LIN {X 0,Y 315.131,Z 1203.889,A -85,B 0,C 180,E1 20783.16,E2 20783.16} C_VEL
LIN {X 0,Y 315.154,Z 1205.25,A -85,B 0,C 180,E1 20791.453,E2 20791.453} C_VEL
LIN {X 0,Y 316.158,Z 1199.354,A -85,B 0,C 180,E1 20803.96,E2 20803.96} C_VEL
LIN {X 0,Y 324.048,Z 1181.565,A -85,B 0,C 180,E1 20817.292,E2 20817.292} C_VEL
LIN {X 0,Y 343.7,Z 1149.442,A -85,B 0,C 180,E1 20829.889,E2 20829.889} C_VEL
LIN {X 0,Y 371.507,Z 1103.542,A -85,B 0,C 180,E1 20840.099,E2 20840.099} C_VEL
LIN {X 0,Y 400.716,Z 1046.598,A -85,B 0,C 180,E1 20847.513,E2 20847.513} C_VEL
LIN {X 0,Y 425.345,Z 983.768,A -85,B 0,C 180,E1 20852.408,E2 20852.408} C_VEL
LIN {X 0,Y 433.911,Z 955.043,A -85,B 0,C 180,E1 20854.017,E2 20854.017} C_VEL
LIN {X 0,Y 421.498,Z 919.963,A -85,B 0,C 180,E1 20862.12,E2 20862.12} C_VEL
LIN {X 0,Y 420.35,Z 917.292,A -85,B 0,C 180,E1 20862.934,E2 20862.934} C_VEL
LIN {X 0,Y 411.814,Z 911.622,A -85,B 0,C 180,E1 20867.638,E2 20867.638} C_VEL
LIN {X 0,Y 405.611,Z 896.607,A -85,B 0,C 180,E1 20876.721,E2 20876.721} C_VEL
LIN {X 0,Y 405.544,Z 892.791,A -85,B 0,C 180,E1 20883.154,E2 20883.154} C_VEL
LIN {X 0,Y 410.311,Z 905.519,A -85,B 0,C 180,E1 20893.279,E2 20893.279} C_VEL
LIN {X 0,Y 418.579,Z 929.23,A -85,B 0,C 180,E1 20901.755,E2 20901.755} C_VEL
LIN {X 0,Y 422.011,Z 951.384,A -85,B 0,C 180,E1 20906.592,E2 20906.592} C_VEL
LIN {X 0,Y 394.355,Z 1017.185,A -85,B 0,C 180,E1 20911.799,E2 20911.799} C_VEL
LIN {X 0,Y 362.549,Z 1077.585,A -85,B 0,C 180,E1 20919.822,E2 20919.822} C_VEL
LIN {X 0,Y 334.565,Z 1125.328,A -85,B 0,C 180,E1 20930.491,E2 20930.491} C_VEL
LIN {X 0,Y 315.72,Z 1159.766,A -85,B 0,C 180,E1 20943.524,E2 20943.524} C_VEL
LIN {X 0,Y 308.132,Z 1178.996,A -85,B 0,C 180,E1 20957.121,E2 20957.121} C_VEL
LIN {X 0,Y 307.029,Z 1184.767,A -85,B 0,C 180,E1 20968.509,E2 20968.509} C_VEL
LIN {X 0,Y 307.704,Z 1181.392,A -85,B 0,C 180,E1 20979.862,E2 20979.862} C_VEL
LIN {X 0,Y 313.175,Z 1165.32,A -85,B 0,C 180,E1 20993.345,E2 20993.345} C_VEL
LIN {X 0,Y 330.014,Z 1133.188,A -85,B 0,C 180,E1 21006.999,E2 21006.999} C_VEL
LIN {X 0,Y 356.224,Z 1088.459,A -85,B 0,C 180,E1 21018.097,E2 21018.097} C_VEL
LIN {X 0,Y 357.572,Z 1084.641,A -85,B 0,C 180,E1 21018.97,E2 21018.97} C_VEL
LIN {X 0,Y 328.069,Z 1088.331,A -85,B 0,C 180,E1 21024.778,E2 21024.778} C_VEL
LIN {X 0,Y 313.608,Z 1088.004,A -85,B 0,C 180,E1 21030.075,E2 21030.075} C_VEL
LIN {X 0,Y 311.553,Z 1108.151,A -85,B 0,C 180,E1 21037.077,E2 21037.077} C_VEL
LIN {X 0,Y 312.349,Z 1113.298,A -85,B 0,C 180,E1 21044.589,E2 21044.589} C_VEL
LIN {X 0,Y 315.942,Z 1103.128,A -85,B 0,C 180,E1 21051.839,E2 21051.839} C_VEL
LIN {X 0,Y 320.96,Z 1077.982,A -85,B 0,C 180,E1 21058.088,E2 21058.088} C_VEL
LIN {X 0,Y 326.7,Z 1042.871,A -85,B 0,C 180,E1 21062.595,E2 21062.595} C_VEL
LIN {X 0,Y 356.77,Z 1008.219,A -85,B 0,C 180,E1 21067.385,E2 21067.385} C_VEL
LIN {X 0,Y 393.256,Z 951.699,A -85,B 0,C 180,E1 21071.07,E2 21071.07} C_VEL
LIN {X 0,Y 411.965,Z 913.023,A -85,B 0,C 180,E1 21072.823,E2 21072.823} C_VEL
LIN {X 0,Y 423.19,Z 942.489,A -85,B 0,C 180,E1 21081.626,E2 21081.626} C_VEL
LIN {X 0,Y 427.875,Z 961.762,A -85,B 0,C 180,E1 21085.399,E2 21085.399} C_VEL
LIN {X 0,Y 404.101,Z 1028.215,A -85,B 0,C 180,E1 21089.854,E2 21089.854} C_VEL
LIN {X 0,Y 375.524,Z 1086.146,A -85,B 0,C 180,E1 21096.292,E2 21096.292} C_VEL
LIN {X 0,Y 346.004,Z 1135.355,A -85,B 0,C 180,E1 21105.534,E2 21105.534} C_VEL
LIN {X 0,Y 322.579,Z 1171.597,A -85,B 0,C 180,E1 21117.338,E2 21117.338} C_VEL
LIN {X 0,Y 310.478,Z 1193.301,A -85,B 0,C 180,E1 21130.074,E2 21130.074} C_VEL
LIN {X 0,Y 307.152,Z 1203.616,A -85,B 0,C 180,E1 21142.982,E2 21142.982} C_VEL
LIN {X 0,Y 307.154,Z 1204.986,A -85,B 0,C 180,E1 21151.49,E2 21151.49} C_VEL
LIN {X 0,Y 308.235,Z 1199.058,A -85,B 0,C 180,E1 21164.326,E2 21164.326} C_VEL
LIN {X 0,Y 316.646,Z 1181.267,A -85,B 0,C 180,E1 21177.936,E2 21177.936} C_VEL
LIN {X 0,Y 337.284,Z 1148.896,A -85,B 0,C 180,E1 21190.806,E2 21190.806} C_VEL
LIN {X 0,Y 365.305,Z 1104.183,A -85,B 0,C 180,E1 21200.884,E2 21200.884} C_VEL
LIN {X 0,Y 395.451,Z 1047.578,A -85,B 0,C 180,E1 21208.369,E2 21208.369} C_VEL
LIN {X 0,Y 421.317,Z 983.665,A -85,B 0,C 180,E1 21213.363,E2 21213.363} C_VEL
LIN {X 0,Y 428.388,Z 957.756,A -85,B 0,C 180,E1 21215.019,E2 21215.019} C_VEL
LIN {X 0,Y 416.291,Z 922.873,A -85,B 0,C 180,E1 21223.622,E2 21223.622} C_VEL
LIN {X 0,Y 411.814,Z 911.622,A -85,B 0,C 180,E1 21227.638,E2 21227.638} C_VEL
LIN {X 0,Y 405.086,Z 909.3,A -85,B 0,C 180,E1 21232.543,E2 21232.543} C_VEL
LIN {X 0,Y 402.968,Z 900.428,A -85,B 0,C 180,E1 21243.174,E2 21243.174} C_VEL
LIN {X 0,Y 407.499,Z 913.449,A -85,B 0,C 180,E1 21253.392,E2 21253.392} C_VEL
LIN {X 0,Y 414.782,Z 936.697,A -85,B 0,C 180,E1 21261.671,E2 21261.671} C_VEL
LIN {X 0,Y 416.844,Z 956.153,A -85,B 0,C 180,E1 21265.866,E2 21265.866} C_VEL
LIN {X 0,Y 388.043,Z 1021.702,A -85,B 0,C 180,E1 21271.213,E2 21271.213} C_VEL
LIN {X 0,Y 356.34,Z 1079.599,A -85,B 0,C 180,E1 21279.086,E2 21279.086} C_VEL
LIN {X 0,Y 326.739,Z 1127.976,A -85,B 0,C 180,E1 21290.237,E2 21290.237} C_VEL
LIN {X 0,Y 307.623,Z 1161.365,A -85,B 0,C 180,E1 21303.562,E2 21303.562} C_VEL
LIN {X 0,Y 300.218,Z 1179.27,A -85,B 0,C 180,E1 21316.775,E2 21316.775} C_VEL
LIN {X 0,Y 299.031,Z 1185.03,A -85,B 0,C 180,E1 21328.469,E2 21328.469} C_VEL
LIN {X 0,Y 299.733,Z 1181.663,A -85,B 0,C 180,E1 21340.127,E2 21340.127} C_VEL
LIN {X 0,Y 305.639,Z 1165.65,A -85,B 0,C 180,E1 21353.93,E2 21353.93} C_VEL
LIN {X 0,Y 323.692,Z 1133.18,A -85,B 0,C 180,E1 21367.991,E2 21367.991} C_VEL
LIN {X 0,Y 349.387,Z 1090.484,A -85,B 0,C 180,E1 21378.869,E2 21378.869} C_VEL
LIN {X 0,Y 315.361,Z 1093.317,A -85,B 0,C 180,E1 21386.504,E2 21386.504} C_VEL
LIN {X 0,Y 305.321,Z 1093.594,A -85,B 0,C 180,E1 21391.106,E2 21391.106} C_VEL
LIN {X 0,Y 303.549,Z 1110.784,A -85,B 0,C 180,E1 21398.074,E2 21398.074} C_VEL
LIN {X 0,Y 304.837,Z 1114.039,A -85,B 0,C 180,E1 21405.765,E2 21405.765} C_VEL
LIN {X 0,Y 308.957,Z 1102.249,A -85,B 0,C 180,E1 21413.031,E2 21413.031} C_VEL
LIN {X 0,Y 314.302,Z 1075.933,A -85,B 0,C 180,E1 21419.217,E2 21419.217} C_VEL
LIN {X 0,Y 318.593,Z 1052.265,A -85,B 0,C 180,E1 21422.496,E2 21422.496} C_VEL
LIN {X 0,Y 348.177,Z 1021.018,A -85,B 0,C 180,E1 21427.627,E2 21427.627} C_VEL
LIN {X 0,Y 387.366,Z 966.083,A -85,B 0,C 180,E1 21431.617,E2 21431.617} C_VEL
LIN {X 0,Y 410.03,Z 922.736,A -85,B 0,C 180,E1 21433.707,E2 21433.707} C_VEL
LIN {X 0,Y 420.798,Z 954.604,A -85,B 0,C 180,E1 21442.592,E2 21442.592} C_VEL
LIN {X 0,Y 422.833,Z 965.85,A -85,B 0,C 180,E1 21444.637,E2 21444.637} C_VEL
LIN {X 0,Y 397.487,Z 1032.998,A -85,B 0,C 180,E1 21449.295,E2 21449.295} C_VEL
LIN {X 0,Y 367.249,Z 1091.263,A -85,B 0,C 180,E1 21456.091,E2 21456.091} C_VEL
LIN {X 0,Y 336.743,Z 1139.701,A -85,B 0,C 180,E1 21465.796,E2 21465.796} C_VEL
LIN {X 0,Y 313.19,Z 1174.637,A -85,B 0,C 180,E1 21478.126,E2 21478.126} C_VEL
LIN {X 0,Y 301.461,Z 1195.76,A -85,B 0,C 180,E1 21492.07,E2 21492.07} C_VEL
LIN {X 0,Y 299.108,Z 1204.275,A -85,B 0,C 180,E1 21505.713,E2 21505.713} C_VEL
LIN {X 0,Y 299.153,Z 1203.069,A -85,B 0,C 180,E1 21517.906,E2 21517.906} C_VEL
LIN {X 0,Y 303.852,Z 1190.722,A -85,B 0,C 180,E1 21532.295,E2 21532.295} C_VEL
LIN {X 0,Y 320.169,Z 1164.103,A -85,B 0,C 180,E1 21546.417,E2 21546.417} C_VEL
LIN {X 0,Y 346.421,Z 1124.982,A -85,B 0,C 180,E1 21557.756,E2 21557.756} C_VEL
LIN {X 0,Y 376.502,Z 1074.926,A -85,B 0,C 180,E1 21566.192,E2 21566.192} C_VEL
LIN {X 0,Y 405.351,Z 1014.417,A -85,B 0,C 180,E1 21572.292,E2 21572.292} C_VEL
LIN {X 0,Y 423.592,Z 962.674,A -85,B 0,C 180,E1 21575.609,E2 21575.609} C_VEL
LIN {X 0,Y 412.761,Z 929.669,A -85,B 0,C 180,E1 21583.933,E2 21583.933} C_VEL
LIN {X 0,Y 405.086,Z 909.3,A -85,B 0,C 180,E1 21592.543,E2 21592.543} C_VEL
LIN {X 0,Y 400.156,Z 911.018,A -85,B 0,C 180,E1 21597.565,E2 21597.565} C_VEL
LIN {X 0,Y 400.518,Z 908.117,A -85,B 0,C 180,E1 21603.194,E2 21603.194} C_VEL
LIN {X 0,Y 404.248,Z 920.191,A -85,B 0,C 180,E1 21612.95,E2 21612.95} C_VEL
LIN {X 0,Y 410.57,Z 942.627,A -85,B 0,C 180,E1 21621.209,E2 21621.209} C_VEL
LIN {X 0,Y 412.177,Z 959.739,A -85,B 0,C 180,E1 21625.055,E2 21625.055} C_VEL
LIN {X 0,Y 382.094,Z 1025.525,A -85,B 0,C 180,E1 21630.529,E2 21630.529} C_VEL
LIN {X 0,Y 348.928,Z 1083.517,A -85,B 0,C 180,E1 21638.686,E2 21638.686} C_VEL
LIN {X 0,Y 318.994,Z 1130.538,A -85,B 0,C 180,E1 21649.954,E2 21649.954} C_VEL
LIN {X 0,Y 299.513,Z 1162.965,A -85,B 0,C 180,E1 21663.601,E2 21663.601} C_VEL
LIN {X 0,Y 292.316,Z 1179.544,A -85,B 0,C 180,E1 21676.411,E2 21676.411} C_VEL
LIN {X 0,Y 291.041,Z 1185.293,A -85,B 0,C 180,E1 21688.427,E2 21688.427} C_VEL
LIN {X 0,Y 291.769,Z 1181.936,A -85,B 0,C 180,E1 21700.407,E2 21700.407} C_VEL
LIN {X 0,Y 297.561,Z 1166.965,A -85,B 0,C 180,E1 21713.902,E2 21713.902} C_VEL
LIN {X 0,Y 315.642,Z 1135.83,A -85,B 0,C 180,E1 21728.142,E2 21728.142} C_VEL
LIN {X 0,Y 339.978,Z 1096.243,A -85,B 0,C 180,E1 21738.919,E2 21738.919} C_VEL
LIN {X 0,Y 310.182,Z 1098.354,A -85,B 0,C 180,E1 21745.869,E2 21745.869} C_VEL
LIN {X 0,Y 296.873,Z 1098.049,A -85,B 0,C 180,E1 21752.042,E2 21752.042} C_VEL
LIN {X 0,Y 295.59,Z 1112.991,A -85,B 0,C 180,E1 21759.035,E2 21759.035} C_VEL
LIN {X 0,Y 297.337,Z 1114.841,A -85,B 0,C 180,E1 21766.813,E2 21766.813} C_VEL
LIN {X 0,Y 302.125,Z 1101.315,A -85,B 0,C 180,E1 21774.32,E2 21774.32} C_VEL
LIN {X 0,Y 307.885,Z 1073.731,A -85,B 0,C 180,E1 21780.436,E2 21780.436} C_VEL
LIN {X 0,Y 311.61,Z 1060.112,A -85,B 0,C 180,E1 21782.66,E2 21782.66} C_VEL
LIN {X 0,Y 343.879,Z 1028.138,A -85,B 0,C 180,E1 21788.412,E2 21788.412} C_VEL
LIN {X 0,Y 384.153,Z 974.953,A -85,B 0,C 180,E1 21792.405,E2 21792.405} C_VEL
LIN {X 0,Y 407.556,Z 932.261,A -85,B 0,C 180,E1 21794.343,E2 21794.343} C_VEL
LIN {X 0,Y 417.432,Z 963.741,A -85,B 0,C 180,E1 21802.883,E2 21802.883} C_VEL
LIN {X 0,Y 417.409,Z 971.066,A -85,B 0,C 180,E1 21803.924,E2 21803.924} C_VEL
LIN {X 0,Y 390.801,Z 1037.652,A -85,B 0,C 180,E1 21808.729,E2 21808.729} C_VEL
LIN {X 0,Y 359.742,Z 1094.763,A -85,B 0,C 180,E1 21815.667,E2 21815.667} C_VEL
LIN {X 0,Y 328.906,Z 1141.72,A -85,B 0,C 180,E1 21825.471,E2 21825.471} C_VEL
LIN {X 0,Y 304.384,Z 1176.732,A -85,B 0,C 180,E1 21838.527,E2 21838.527} C_VEL
LIN {X 0,Y 293.483,Z 1195.888,A -85,B 0,C 180,E1 21852.011,E2 21852.011} C_VEL
LIN {X 0,Y 291.097,Z 1204.007,A -85,B 0,C 180,E1 21865.595,E2 21865.595} C_VEL
LIN {X 0,Y 291.163,Z 1203.01,A -85,B 0,C 180,E1 21877.566,E2 21877.566} C_VEL
LIN {X 0,Y 295.159,Z 1192.452,A -85,B 0,C 180,E1 21891.175,E2 21891.175} C_VEL
LIN {X 0,Y 310.316,Z 1168.09,A -85,B 0,C 180,E1 21905.499,E2 21905.499} C_VEL
LIN {X 0,Y 337.055,Z 1129.942,A -85,B 0,C 180,E1 21917.545,E2 21917.545} C_VEL
LIN {X 0,Y 368.849,Z 1079.537,A -85,B 0,C 180,E1 21926.579,E2 21926.579} C_VEL
LIN {X 0,Y 399.806,Z 1017.759,A -85,B 0,C 180,E1 21933.031,E2 21933.031} C_VEL
LIN {X 0,Y 418.696,Z 967.227,A -85,B 0,C 180,E1 21936.303,E2 21936.303} C_VEL
LIN {X 0,Y 408.498,Z 934.625,A -85,B 0,C 180,E1 21944.866,E2 21944.866} C_VEL
LIN {X 0,Y 401.343,Z 913.898,A -85,B 0,C 180,E1 21954.513,E2 21954.513} C_VEL
LIN {X 0,Y 400.156,Z 911.018,A -85,B 0,C 180,E1 21957.565,E2 21957.565} C_VEL
LIN {X 0,Y 397.67,Z 915.644,A -85,B 0,C 180,E1 21962.65,E2 21962.65} C_VEL
LIN {X 0,Y 400.781,Z 926.844,A -85,B 0,C 180,E1 21972.508,E2 21972.508} C_VEL
LIN {X 0,Y 406.304,Z 948.436,A -85,B 0,C 180,E1 21980.711,E2 21980.711} C_VEL
LIN {X 0,Y 407.109,Z 964.414,A -85,B 0,C 180,E1 21984.297,E2 21984.297} C_VEL
LIN {X 0,Y 375.809,Z 1030.127,A -85,B 0,C 180,E1 21989.909,E2 21989.909} C_VEL
LIN {X 0,Y 341.819,Z 1086.973,A -85,B 0,C 180,E1 21998.178,E2 21998.178} C_VEL
LIN {X 0,Y 311.225,Z 1132.932,A -85,B 0,C 180,E1 22009.663,E2 22009.663} C_VEL
LIN {X 0,Y 291.412,Z 1164.556,A -85,B 0,C 180,E1 22023.643,E2 22023.643} C_VEL
LIN {X 0,Y 284.061,Z 1181.005,A -85,B 0,C 180,E1 22037.58,E2 22037.58} C_VEL
LIN {X 0,Y 283.042,Z 1185.556,A -85,B 0,C 180,E1 22048.383,E2 22048.383} C_VEL
LIN {X 0,Y 283.837,Z 1182.208,A -85,B 0,C 180,E1 22060.701,E2 22060.701} C_VEL
LIN {X 0,Y 290.254,Z 1166.966,A -85,B 0,C 180,E1 22074.758,E2 22074.758} C_VEL
LIN {X 0,Y 309.907,Z 1135.149,A -85,B 0,C 180,E1 22089.434,E2 22089.434} C_VEL
LIN {X 0,Y 331.577,Z 1102.546,A -85,B 0,C 180,E1 22098.535,E2 22098.535} C_VEL
LIN {X 0,Y 292.123,Z 1101.841,A -85,B 0,C 180,E1 22110.535,E2 22110.535} C_VEL
LIN {X 0,Y 288.505,Z 1102.454,A -85,B 0,C 180,E1 22113.114,E2 22113.114} C_VEL
LIN {X 0,Y 287.724,Z 1115.062,A -85,B 0,C 180,E1 22120.049,E2 22120.049} C_VEL
LIN {X 0,Y 289.979,Z 1115.281,A -85,B 0,C 180,E1 22128.009,E2 22128.009} C_VEL
LIN {X 0,Y 295.095,Z 1101.275,A -85,B 0,C 180,E1 22135.294,E2 22135.294} C_VEL
LIN {X 0,Y 301.281,Z 1073.043,A -85,B 0,C 180,E1 22141.443,E2 22141.443} C_VEL
LIN {X 0,Y 332.801,Z 1041.917,A -85,B 0,C 180,E1 22148.307,E2 22148.307} C_VEL
LIN {X 0,Y 370.527,Z 998.297,A -85,B 0,C 180,E1 22152.317,E2 22152.317} C_VEL
LIN {X 0,Y 405.129,Z 942.403,A -85,B 0,C 180,E1 22155.152,E2 22155.152} C_VEL
LIN {X 0,Y 413.383,Z 971.51,A -85,B 0,C 180,E1 22162.877,E2 22162.877} C_VEL
LIN {X 0,Y 385.674,Z 1039.157,A -85,B 0,C 180,E1 22167.852,E2 22167.852} C_VEL
LIN {X 0,Y 353.683,Z 1095.936,A -85,B 0,C 180,E1 22174.854,E2 22174.854} C_VEL
LIN {X 0,Y 321.493,Z 1143.165,A -85,B 0,C 180,E1 22184.97,E2 22184.97} C_VEL
LIN {X 0,Y 297.302,Z 1176.315,A -85,B 0,C 180,E1 22197.688,E2 22197.688} C_VEL
LIN {X 0,Y 285.69,Z 1195.579,A -85,B 0,C 180,E1 22211.503,E2 22211.503} C_VEL
LIN {X 0,Y 283.086,Z 1203.74,A -85,B 0,C 180,E1 22225.47,E2 22225.47} C_VEL
LIN {X 0,Y 283.16,Z 1202.736,A -85,B 0,C 180,E1 22237.781,E2 22237.781} C_VEL
LIN {X 0,Y 287.881,Z 1191.263,A -85,B 0,C 180,E1 22252.502,E2 22252.502} C_VEL
LIN {X 0,Y 304.932,Z 1165.727,A -85,B 0,C 180,E1 22267.258,E2 22267.258} C_VEL
LIN {X 0,Y 333.289,Z 1126.674,A -85,B 0,C 180,E1 22279.271,E2 22279.271} C_VEL
LIN {X 0,Y 366.462,Z 1074.958,A -85,B 0,C 180,E1 22288.201,E2 22288.201} C_VEL
LIN {X 0,Y 397.562,Z 1013.386,A -85,B 0,C 180,E1 22294.377,E2 22294.377} C_VEL
LIN {X 0,Y 413.495,Z 970.598,A -85,B 0,C 180,E1 22297.272,E2 22297.272} C_VEL
LIN {X 0,Y 404.379,Z 939.598,A -85,B 0,C 180,E1 22305.819,E2 22305.819} C_VEL
LIN {X 0,Y 398.564,Z 921.554,A -85,B 0,C 180,E1 22314.475,E2 22314.475} C_VEL
LIN {X 0,Y 397.67,Z 915.644,A -85,B 0,C 180,E1 22322.65,E2 22322.65} C_VEL
LIN {X 0,Y 395.493,Z 927.102,A -85,B 0,C 180,E1 22327.511,E2 22327.511} C_VEL
LIN {X 0,Y 399.893,Z 943.083,A -85,B 0,C 180,E1 22336.466,E2 22336.466} C_VEL
LIN {X 0,Y 403.092,Z 966.647,A -85,B 0,C 180,E1 22343.368,E2 22343.368} C_VEL
LIN {X 0,Y 370.657,Z 1032.667,A -85,B 0,C 180,E1 22349.043,E2 22349.043} C_VEL
LIN {X 0,Y 334.918,Z 1090.181,A -85,B 0,C 180,E1 22357.608,E2 22357.608} C_VEL
LIN {X 0,Y 303.466,Z 1135.317,A -85,B 0,C 180,E1 22369.358,E2 22369.358} C_VEL
LIN {X 0,Y 283.284,Z 1166.142,A -85,B 0,C 180,E1 22383.685,E2 22383.685} C_VEL
LIN {X 0,Y 276.141,Z 1181.277,A -85,B 0,C 180,E1 22397.218,E2 22397.218} C_VEL
LIN {X 0,Y 275.061,Z 1185.818,A -85,B 0,C 180,E1 22408.336,E2 22408.336} C_VEL
LIN {X 0,Y 275.88,Z 1182.482,A -85,B 0,C 180,E1 22421.013,E2 22421.013} C_VEL
LIN {X 0,Y 283.386,Z 1166.245,A -85,B 0,C 180,E1 22436.124,E2 22436.124} C_VEL
LIN {X 0,Y 304.985,Z 1133.458,A -85,B 0,C 180,E1 22451.139,E2 22451.139} C_VEL
LIN {X 0,Y 322.454,Z 1107.331,A -85,B 0,C 180,E1 22458.725,E2 22458.725} C_VEL
LIN {X 0,Y 286.524,Z 1106.683,A -85,B 0,C 180,E1 22469.9,E2 22469.9} C_VEL
LIN {X 0,Y 280.225,Z 1106.965,A -85,B 0,C 180,E1 22474.433,E2 22474.433} C_VEL
LIN {X 0,Y 280.213,Z 1117.935,A -85,B 0,C 180,E1 22482.769,E2 22482.769} C_VEL
LIN {X 0,Y 283.83,Z 1113.485,A -85,B 0,C 180,E1 22490.96,E2 22490.96} C_VEL
LIN {X 0,Y 289.866,Z 1094.829,A -85,B 0,C 180,E1 22498.144,E2 22498.144} C_VEL
LIN {X 0,Y 295.732,Z 1076.127,A -85,B 0,C 180,E1 22502.379,E2 22502.379} C_VEL
LIN {X 0,Y 328.939,Z 1047.886,A -85,B 0,C 180,E1 22509.156,E2 22509.156} C_VEL
LIN {X 0,Y 367.954,Z 1005.018,A -85,B 0,C 180,E1 22513.256,E2 22513.256} C_VEL
LIN {X 0,Y 401.627,Z 953.589,A -85,B 0,C 180,E1 22515.766,E2 22515.766} C_VEL
LIN {X 0,Y 408.449,Z 975.566,A -85,B 0,C 180,E1 22522.058,E2 22522.058} C_VEL
LIN {X 0,Y 379.632,Z 1042.643,A -85,B 0,C 180,E1 22527.148,E2 22527.148} C_VEL
LIN {X 0,Y 345.909,Z 1099.798,A -85,B 0,C 180,E1 22534.455,E2 22534.455} C_VEL
LIN {X 0,Y 313.362,Z 1145.403,A -85,B 0,C 180,E1 22544.708,E2 22544.708} C_VEL
LIN {X 0,Y 288.225,Z 1178.628,A -85,B 0,C 180,E1 22558.329,E2 22558.329} C_VEL
LIN {X 0,Y 276.792,Z 1197.798,A -85,B 0,C 180,E1 22573.921,E2 22573.921} C_VEL
LIN {X 0,Y 275.444,Z 1203.953,A -85,B 0,C 180,E1 22588.505,E2 22588.505} C_VEL
LIN {X 0,Y 275.544,Z 1200.991,A -85,B 0,C 180,E1 22601.198,E2 22601.198} C_VEL
LIN {X 0,Y 282.606,Z 1186.833,A -85,B 0,C 180,E1 22616.383,E2 22616.383} C_VEL
LIN {X 0,Y 302.705,Z 1159.411,A -85,B 0,C 180,E1 22630.569,E2 22630.569} C_VEL
LIN {X 0,Y 333.514,Z 1118.043,A -85,B 0,C 180,E1 22642.14,E2 22642.14} C_VEL
LIN {X 0,Y 367.99,Z 1064.17,A -85,B 0,C 180,E1 22650.58,E2 22650.58} C_VEL
LIN {X 0,Y 399.257,Z 1000.706,A -85,B 0,C 180,E1 22656.295,E2 22656.295} C_VEL
LIN {X 0,Y 408.754,Z 975.453,A -85,B 0,C 180,E1 22657.911,E2 22657.911} C_VEL
LIN {X 0,Y 400.47,Z 944.955,A -85,B 0,C 180,E1 22666.647,E2 22666.647} C_VEL
LIN {X 0,Y 395.299,Z 927.991,A -85,B 0,C 180,E1 22675.533,E2 22675.533} C_VEL
LIN {X 0,Y 395.076,Z 923.298,A -85,B 0,C 180,E1 22683.238,E2 22683.238} C_VEL
LIN {X 0,Y 395.493,Z 927.102,A -85,B 0,C 180,E1 22687.511,E2 22687.511} C_VEL
LIN {X 0,Y 394.052,Z 941.312,A -85,B 0,C 180,E1 22692.253,E2 22692.253} C_VEL
LIN {X 0,Y 397.916,Z 962.413,A -85,B 0,C 180,E1 22700.401,E2 22700.401} C_VEL
LIN {X 0,Y 397.294,Z 973.158,A -85,B 0,C 180,E1 22702.704,E2 22702.704} C_VEL
LIN {X 0,Y 365.151,Z 1035.888,A -85,B 0,C 180,E1 22708.234,E2 22708.234} C_VEL
LIN {X 0,Y 328.089,Z 1093.249,A -85,B 0,C 180,E1 22716.98,E2 22716.98} C_VEL
LIN {X 0,Y 295.686,Z 1137.76,A -85,B 0,C 180,E1 22729.065,E2 22729.065} C_VEL
LIN {X 0,Y 275.159,Z 1167.655,A -85,B 0,C 180,E1 22743.729,E2 22743.729} C_VEL
LIN {X 0,Y 267.913,Z 1182.72,A -85,B 0,C 180,E1 22758.479,E2 22758.479} C_VEL
LIN {X 0,Y 267.305,Z 1186.081,A -85,B 0,C 180,E1 22771.54,E2 22771.54} C_VEL
LIN {X 0,Y 268.748,Z 1180.419,A -85,B 0,C 180,E1 22784.63,E2 22784.63} C_VEL
LIN {X 0,Y 279.144,Z 1161.673,A -85,B 0,C 180,E1 22799.908,E2 22799.908} C_VEL
LIN {X 0,Y 304.13,Z 1126.199,A -85,B 0,C 180,E1 22814.698,E2 22814.698} C_VEL
LIN {X 0,Y 313.78,Z 1112.947,A -85,B 0,C 180,E1 22818.439,E2 22818.439} C_VEL
LIN {X 0,Y 273.149,Z 1109.843,A -85,B 0,C 180,E1 22833.933,E2 22833.933} C_VEL
LIN {X 0,Y 272.175,Z 1118.664,A -85,B 0,C 180,E1 22842.244,E2 22842.244} C_VEL
LIN {X 0,Y 275.749,Z 1115.841,A -85,B 0,C 180,E1 22850.693,E2 22850.693} C_VEL
LIN {X 0,Y 282.175,Z 1098.558,A -85,B 0,C 180,E1 22858.22,E2 22858.22} C_VEL
LIN {X 0,Y 288.684,Z 1082.785,A -85,B 0,C 180,E1 22862.437,E2 22862.437} C_VEL
LIN {X 0,Y 320.525,Z 1057.611,A -85,B 0,C 180,E1 22869.384,E2 22869.384} C_VEL
LIN {X 0,Y 359.428,Z 1018.698,A -85,B 0,C 180,E1 22873.703,E2 22873.703} C_VEL
LIN {X 0,Y 399.535,Z 962.43,A -85,B 0,C 180,E1 22876.614,E2 22876.614} C_VEL
LIN {X 0,Y 403.018,Z 981.793,A -85,B 0,C 180,E1 22881.461,E2 22881.461} C_VEL
LIN {X 0,Y 373.068,Z 1047.004,A -85,B 0,C 180,E1 22886.506,E2 22886.506} C_VEL
LIN {X 0,Y 338.243,Z 1103.455,A -85,B 0,C 180,E1 22894.034,E2 22894.034} C_VEL
LIN {X 0,Y 304.321,Z 1148.9,A -85,B 0,C 180,E1 22904.832,E2 22904.832} C_VEL
LIN {X 0,Y 279.168,Z 1180.87,A -85,B 0,C 180,E1 22919.009,E2 22919.009} C_VEL
LIN {X 0,Y 268.913,Z 1197.494,A -85,B 0,C 180,E1 22933.436,E2 22933.436} C_VEL
LIN {X 0,Y 267.427,Z 1203.689,A -85,B 0,C 180,E1 22948.461,E2 22948.461} C_VEL
LIN {X 0,Y 267.576,Z 1200.713,A -85,B 0,C 180,E1 22961.536,E2 22961.536} C_VEL
LIN {X 0,Y 275.195,Z 1186.491,A -85,B 0,C 180,E1 22977.151,E2 22977.151} C_VEL
LIN {X 0,Y 296.549,Z 1158.675,A -85,B 0,C 180,E1 22991.736,E2 22991.736} C_VEL
LIN {X 0,Y 328.368,Z 1117.393,A -85,B 0,C 180,E1 23003.311,E2 23003.311} C_VEL
LIN {X 0,Y 363.512,Z 1064.027,A -85,B 0,C 180,E1 23011.658,E2 23011.658} C_VEL
LIN {X 0,Y 395.166,Z 1001.593,A -85,B 0,C 180,E1 23017.278,E2 23017.278} C_VEL
LIN {X 0,Y 403.746,Z 979.378,A -85,B 0,C 180,E1 23018.769,E2 23018.769} C_VEL
LIN {X 0,Y 396.717,Z 951.252,A -85,B 0,C 180,E1 23027.156,E2 23027.156} C_VEL
LIN {X 0,Y 392.394,Z 935.531,A -85,B 0,C 180,E1 23035.5,E2 23035.5} C_VEL
LIN {X 0,Y 391.999,Z 930.761,A -85,B 0,C 180,E1 23043.263,E2 23043.263} C_VEL
LIN {X 0,Y 394.052,Z 941.312,A -85,B 0,C 180,E1 23052.253,E2 23052.253} C_VEL
LIN {X 0,Y 392.449,Z 958.805,A -85,B 0,C 180,E1 23056.783,E2 23056.783} C_VEL
LIN {X 0,Y 393.029,Z 976.289,A -85,B 0,C 180,E1 23061.801,E2 23061.801} C_VEL
LIN {X 0,Y 359.901,Z 1038.703,A -85,B 0,C 180,E1 23067.365,E2 23067.365} C_VEL
LIN {X 0,Y 322.167,Z 1095.067,A -85,B 0,C 180,E1 23076.091,E2 23076.091} C_VEL
LIN {X 0,Y 287.97,Z 1140.055,A -85,B 0,C 180,E1 23088.698,E2 23088.698} C_VEL
LIN {X 0,Y 267.037,Z 1169.05,A -85,B 0,C 180,E1 23103.777,E2 23103.777} C_VEL
LIN {X 0,Y 259.976,Z 1182.992,A -85,B 0,C 180,E1 23118.122,E2 23118.122} C_VEL
LIN {X 0,Y 259.301,Z 1186.345,A -85,B 0,C 180,E1 23131.588,E2 23131.588} C_VEL
LIN {X 0,Y 260.894,Z 1180.7,A -85,B 0,C 180,E1 23145.08,E2 23145.08} C_VEL
LIN {X 0,Y 271.951,Z 1161.987,A -85,B 0,C 180,E1 23160.784,E2 23160.784} C_VEL
LIN {X 0,Y 298.227,Z 1126.567,A -85,B 0,C 180,E1 23175.833,E2 23175.833} C_VEL
LIN {X 0,Y 304.96,Z 1116.771,A -85,B 0,C 180,E1 23178.871,E2 23178.871} C_VEL
LIN {X 0,Y 269.786,Z 1115.228,A -85,B 0,C 180,E1 23191.551,E2 23191.551} C_VEL
LIN {X 0,Y 263.941,Z 1114.097,A -85,B 0,C 180,E1 23197.121,E2 23197.121} C_VEL
LIN {X 0,Y 265.057,Z 1120.602,A -85,B 0,C 180,E1 23205.172,E2 23205.172} C_VEL
LIN {X 0,Y 270.073,Z 1113.446,A -85,B 0,C 180,E1 23213.644,E2 23213.644} C_VEL
LIN {X 0,Y 280.504,Z 1090.001,A -85,B 0,C 180,E1 23222.164,E2 23222.164} C_VEL
LIN {X 0,Y 311.63,Z 1067.113,A -85,B 0,C 180,E1 23229.516,E2 23229.516} C_VEL
LIN {X 0,Y 350.008,Z 1032.217,A -85,B 0,C 180,E1 23234.082,E2 23234.082} C_VEL
LIN {X 0,Y 393.198,Z 977.411,A -85,B 0,C 180,E1 23237.179,E2 23237.179} C_VEL
LIN {X 0,Y 396.123,Z 972.641,A -85,B 0,C 180,E1 23237.336,E2 23237.336} C_VEL
LIN {X 0,Y 397.973,Z 986.103,A -85,B 0,C 180,E1 23240.657,E2 23240.657} C_VEL
LIN {X 0,Y 366.671,Z 1051.009,A -85,B 0,C 180,E1 23245.829,E2 23245.829} C_VEL
LIN {X 0,Y 330.683,Z 1106.725,A -85,B 0,C 180,E1 23253.532,E2 23253.532} C_VEL
LIN {X 0,Y 296.276,Z 1150.88,A -85,B 0,C 180,E1 23264.52,E2 23264.52} C_VEL
LIN {X 0,Y 271.065,Z 1181.72,A -85,B 0,C 180,E1 23278.917,E2 23278.917} C_VEL
LIN {X 0,Y 260.453,Z 1198.551,A -85,B 0,C 180,E1 23294.894,E2 23294.894} C_VEL
LIN {X 0,Y 259.433,Z 1203.425,A -85,B 0,C 180,E1 23308.413,E2 23308.413} C_VEL
LIN {X 0,Y 259.616,Z 1200.423,A -85,B 0,C 180,E1 23321.894,E2 23321.894} C_VEL
LIN {X 0,Y 267.731,Z 1186.249,A -85,B 0,C 180,E1 23337.861,E2 23337.861} C_VEL
LIN {X 0,Y 290.328,Z 1158.17,A -85,B 0,C 180,E1 23352.841,E2 23352.841} C_VEL
LIN {X 0,Y 323.511,Z 1116.592,A -85,B 0,C 180,E1 23364.542,E2 23364.542} C_VEL
LIN {X 0,Y 359.623,Z 1063.18,A -85,B 0,C 180,E1 23372.848,E2 23372.848} C_VEL
LIN {X 0,Y 392.039,Z 1000.643,A -85,B 0,C 180,E1 23378.405,E2 23378.405} C_VEL
LIN {X 0,Y 398.873,Z 983.52,A -85,B 0,C 180,E1 23379.606,E2 23379.606} C_VEL
LIN {X 0,Y 392.607,Z 956.237,A -85,B 0,C 180,E1 23388.171,E2 23388.171} C_VEL
LIN {X 0,Y 388.92,Z 941.933,A -85,B 0,C 180,E1 23396.58,E2 23396.58} C_VEL
LIN {X 0,Y 389.043,Z 938.272,A -85,B 0,C 180,E1 23403.288,E2 23403.288} C_VEL
LIN {X 0,Y 390.835,Z 949.828,A -85,B 0,C 180,E1 23412.831,E2 23412.831} C_VEL
LIN {X 0,Y 392.449,Z 958.805,A -85,B 0,C 180,E1 23416.783,E2 23416.783} C_VEL
LIN {X 0,Y 389.051,Z 974.042,A -85,B 0,C 180,E1 23419.455,E2 23419.455} C_VEL
LIN {X 0,Y 387.7,Z 981.882,A -85,B 0,C 180,E1 23421.038,E2 23421.038} C_VEL
LIN {X 0,Y 352.867,Z 1044.506,A -85,B 0,C 180,E1 23426.835,E2 23426.835} C_VEL
LIN {X 0,Y 314.505,Z 1099.09,A -85,B 0,C 180,E1 23435.654,E2 23435.654} C_VEL
LIN {X 0,Y 279.781,Z 1142.834,A -85,B 0,C 180,E1 23448.531,E2 23448.531} C_VEL
LIN {X 0,Y 258.942,Z 1170.447,A -85,B 0,C 180,E1 23463.83,E2 23463.83} C_VEL
LIN {X 0,Y 252.067,Z 1183.262,A -85,B 0,C 180,E1 23477.744,E2 23477.744} C_VEL
LIN {X 0,Y 251.297,Z 1186.608,A -85,B 0,C 180,E1 23491.638,E2 23491.638} C_VEL
LIN {X 0,Y 253.047,Z 1180.978,A -85,B 0,C 180,E1 23505.56,E2 23505.56} C_VEL
LIN {X 0,Y 264.961,Z 1162.087,A -85,B 0,C 180,E1 23521.83,E2 23521.83} C_VEL
LIN {X 0,Y 292.469,Z 1126.956,A -85,B 0,C 180,E1 23537.006,E2 23537.006} C_VEL
LIN {X 0,Y 295.141,Z 1121.453,A -85,B 0,C 180,E1 23539.1,E2 23539.1} C_VEL
LIN {X 0,Y 263.938,Z 1119.784,A -85,B 0,C 180,E1 23550.861,E2 23550.861} C_VEL
LIN {X 0,Y 255.947,Z 1118.025,A -85,B 0,C 180,E1 23559.271,E2 23559.271} C_VEL
LIN {X 0,Y 258.507,Z 1121.273,A -85,B 0,C 180,E1 23568.246,E2 23568.246} C_VEL
LIN {X 0,Y 264.611,Z 1110.572,A -85,B 0,C 180,E1 23576.399,E2 23576.399} C_VEL
LIN {X 0,Y 271.903,Z 1097.155,A -85,B 0,C 180,E1 23581.693,E2 23581.693} C_VEL
LIN {X 0,Y 303.672,Z 1075.343,A -85,B 0,C 180,E1 23589.783,E2 23589.783} C_VEL
LIN {X 0,Y 342.138,Z 1043.121,A -85,B 0,C 180,E1 23594.624,E2 23594.624} C_VEL
LIN {X 0,Y 388.136,Z 989.54,A -85,B 0,C 180,E1 23597.891,E2 23597.891} C_VEL
LIN {X 0,Y 392.823,Z 983.081,A -85,B 0,C 180,E1 23598.259,E2 23598.259} C_VEL
LIN {X 0,Y 392.753,Z 990.926,A -85,B 0,C 180,E1 23599.871,E2 23599.871} C_VEL
LIN {X 0,Y 360.016,Z 1055.415,A -85,B 0,C 180,E1 23605.173,E2 23605.173} C_VEL
LIN {X 0,Y 323.57,Z 1109.4,A -85,B 0,C 180,E1 23612.909,E2 23612.909} C_VEL
LIN {X 0,Y 288.702,Z 1152.353,A -85,B 0,C 180,E1 23624.018,E2 23624.018} C_VEL
LIN {X 0,Y 262.981,Z 1182.568,A -85,B 0,C 180,E1 23638.819,E2 23638.819} C_VEL
LIN {X 0,Y 252.584,Z 1198.25,A -85,B 0,C 180,E1 23654.411,E2 23654.411} C_VEL
LIN {X 0,Y 251.416,Z 1203.161,A -85,B 0,C 180,E1 23668.363,E2 23668.363} C_VEL
LIN {X 0,Y 251.69,Z 1200.145,A -85,B 0,C 180,E1 23682.275,E2 23682.275} C_VEL
LIN {X 0,Y 260.414,Z 1185.881,A -85,B 0,C 180,E1 23698.731,E2 23698.731} C_VEL
LIN {X 0,Y 283.879,Z 1158.096,A -85,B 0,C 180,E1 23713.845,E2 23713.845} C_VEL
LIN {X 0,Y 317.536,Z 1117.449,A -85,B 0,C 180,E1 23725.475,E2 23725.475} C_VEL
LIN {X 0,Y 354.511,Z 1064.582,A -85,B 0,C 180,E1 23733.802,E2 23733.802} C_VEL
LIN {X 0,Y 387.934,Z 1002.308,A -85,B 0,C 180,E1 23739.381,E2 23739.381} C_VEL
LIN {X 0,Y 393.818,Z 987.409,A -85,B 0,C 180,E1 23740.523,E2 23740.523} C_VEL
LIN {X 0,Y 388.458,Z 961.241,A -85,B 0,C 180,E1 23749.241,E2 23749.241} C_VEL
LIN {X 0,Y 385.619,Z 948.361,A -85,B 0,C 180,E1 23757.679,E2 23757.679} C_VEL
LIN {X 0,Y 385.682,Z 945.608,A -85,B 0,C 180,E1 23763.317,E2 23763.317} C_VEL
LIN {X 0,Y 387.122,Z 957.256,A -85,B 0,C 180,E1 23772.917,E2 23772.917} C_VEL
LIN {X 0,Y 389.051,Z 974.042,A -85,B 0,C 180,E1 23779.455,E2 23779.455} C_VEL
LIN {X 0,Y 385.327,Z 983.053,A -85,B 0,C 180,E1 23780.316,E2 23780.316} C_VEL
LIN {X 0,Y 378.966,Z 994.037,A -85,B 0,C 180,E1 23780.743,E2 23780.743} C_VEL
LIN {X 0,Y 342.783,Z 1054.779,A -85,B 0,C 180,E1 23786.873,E2 23786.873} C_VEL
LIN {X 0,Y 303.83,Z 1106.966,A -85,B 0,C 180,E1 23796.066,E2 23796.066} C_VEL
LIN {X 0,Y 269.364,Z 1148.127,A -85,B 0,C 180,E1 23809.512,E2 23809.512} C_VEL
LIN {X 0,Y 250.074,Z 1173.094,A -85,B 0,C 180,E1 23824.908,E2 23824.908} C_VEL
LIN {X 0,Y 243.529,Z 1185.202,A -85,B 0,C 180,E1 23840.943,E2 23840.943} C_VEL
LIN {X 0,Y 243.311,Z 1186.332,A -85,B 0,C 180,E1 23855.272,E2 23855.272} C_VEL
LIN {X 0,Y 247.719,Z 1176.741,A -85,B 0,C 180,E1 23871.462,E2 23871.462} C_VEL
LIN {X 0,Y 265.023,Z 1153.312,A -85,B 0,C 180,E1 23887.876,E2 23887.876} C_VEL
LIN {X 0,Y 287.466,Z 1125.946,A -85,B 0,C 180,E1 23898.837,E2 23898.837} C_VEL
LIN {X 0,Y 253.564,Z 1123.075,A -85,B 0,C 180,E1 23913.447,E2 23913.447} C_VEL
LIN {X 0,Y 248.204,Z 1120.687,A -85,B 0,C 180,E1 23921.073,E2 23921.073} C_VEL
LIN {X 0,Y 251.383,Z 1122.109,A -85,B 0,C 180,E1 23929.671,E2 23929.671} C_VEL
LIN {X 0,Y 258.897,Z 1109.023,A -85,B 0,C 180,E1 23938.419,E2 23938.419} C_VEL
LIN {X 0,Y 287.729,Z 1088.457,A -85,B 0,C 180,E1 23948.498,E2 23948.498} C_VEL
LIN {X 0,Y 328.357,Z 1058.46,A -85,B 0,C 180,E1 23954.585,E2 23954.585} C_VEL
LIN {X 0,Y 373.884,Z 1012.259,A -85,B 0,C 180,E1 23958.068,E2 23958.068} C_VEL
LIN {X 0,Y 388.142,Z 994.325,A -85,B 0,C 180,E1 23958.981,E2 23958.981} C_VEL
LIN {X 0,Y 353.702,Z 1059.168,A -85,B 0,C 180,E1 23964.431,E2 23964.431} C_VEL
LIN {X 0,Y 316.125,Z 1112.516,A -85,B 0,C 180,E1 23972.355,E2 23972.355} C_VEL
LIN {X 0,Y 280.204,Z 1154.834,A -85,B 0,C 180,E1 23983.861,E2 23983.861} C_VEL
LIN {X 0,Y 254.861,Z 1183.397,A -85,B 0,C 180,E1 23998.711,E2 23998.711} C_VEL
LIN {X 0,Y 244.551,Z 1198.312,A -85,B 0,C 180,E1 24014.467,E2 24014.467} C_VEL
LIN {X 0,Y 243.407,Z 1202.897,A -85,B 0,C 180,E1 24028.309,E2 24028.309} C_VEL
LIN {X 0,Y 243.744,Z 1199.857,A -85,B 0,C 180,E1 24042.682,E2 24042.682} C_VEL
LIN {X 0,Y 252.79,Z 1185.944,A -85,B 0,C 180,E1 24059.302,E2 24059.302} C_VEL
LIN {X 0,Y 277.154,Z 1158.362,A -85,B 0,C 180,E1 24074.75,E2 24074.75} C_VEL
LIN {X 0,Y 312.187,Z 1117.586,A -85,B 0,C 180,E1 24086.595,E2 24086.595} C_VEL
LIN {X 0,Y 349.992,Z 1065.193,A -85,B 0,C 180,E1 24094.888,E2 24094.888} C_VEL
LIN {X 0,Y 384.317,Z 1003.175,A -85,B 0,C 180,E1 24100.43,E2 24100.43} C_VEL
LIN {X 0,Y 388.956,Z 991.404,A -85,B 0,C 180,E1 24101.452,E2 24101.452} C_VEL
LIN {X 0,Y 384.308,Z 966.362,A -85,B 0,C 180,E1 24110.273,E2 24110.273} C_VEL
LIN {X 0,Y 382.129,Z 954.639,A -85,B 0,C 180,E1 24118.796,E2 24118.796} C_VEL
LIN {X 0,Y 382.438,Z 952.996,A -85,B 0,C 180,E1 24123.345,E2 24123.345} C_VEL
LIN {X 0,Y 383.456,Z 965.278,A -85,B 0,C 180,E1 24133.279,E2 24133.279} C_VEL
LIN {X 0,Y 384.01,Z 984.152,A -85,B 0,C 180,E1 24140.033,E2 24140.033} C_VEL
LIN {X 0,Y 378.966,Z 994.037,A -85,B 0,C 180,E1 24140.743,E2 24140.743} C_VEL
LIN {X 0,Y 360.054,Z 1022.968,A -85,B 0,C 180,E1 24141.978,E2 24141.978} C_VEL
LIN {X 0,Y 320.723,Z 1080.459,A -85,B 0,C 180,E1 24149.415,E2 24149.415} C_VEL
LIN {X 0,Y 281.766,Z 1127.575,A -85,B 0,C 180,E1 24160.388,E2 24160.388} C_VEL
LIN {X 0,Y 251.326,Z 1162.487,A -85,B 0,C 180,E1 24175.94,E2 24175.94} C_VEL
LIN {X 0,Y 237.385,Z 1181.493,A -85,B 0,C 180,E1 24193.182,E2 24193.182} C_VEL
LIN {X 0,Y 235.095,Z 1187.134,A -85,B 0,C 180,E1 24208.053,E2 24208.053} C_VEL
LIN {X 0,Y 236.274,Z 1183.848,A -85,B 0,C 180,E1 24222.889,E2 24222.889} C_VEL
LIN {X 0,Y 247.043,Z 1167.741,A -85,B 0,C 180,E1 24240.337,E2 24240.337} C_VEL
LIN {X 0,Y 274.644,Z 1135.595,A -85,B 0,C 180,E1 24256.778,E2 24256.778} C_VEL
LIN {X 0,Y 278.76,Z 1130.041,A -85,B 0,C 180,E1 24258.873,E2 24258.873} C_VEL
LIN {X 0,Y 243.75,Z 1126.251,A -85,B 0,C 180,E1 24276.248,E2 24276.248} C_VEL
LIN {X 0,Y 241.701,Z 1124.21,A -85,B 0,C 180,E1 24286.26,E2 24286.26} C_VEL
LIN {X 0,Y 248.131,Z 1117.592,A -85,B 0,C 180,E1 24295.68,E2 24295.68} C_VEL
LIN {X 0,Y 268.458,Z 1102.24,A -85,B 0,C 180,E1 24305.719,E2 24305.719} C_VEL
LIN {X 0,Y 305.879,Z 1078.379,A -85,B 0,C 180,E1 24313.296,E2 24313.296} C_VEL
LIN {X 0,Y 349.252,Z 1042.587,A -85,B 0,C 180,E1 24317.627,E2 24317.627} C_VEL
LIN {X 0,Y 374.577,Z 1016.288,A -85,B 0,C 180,E1 24319.374,E2 24319.374} C_VEL
LIN {X 0,Y 337.544,Z 1077.487,A -85,B 0,C 180,E1 24325.453,E2 24325.453} C_VEL
LIN {X 0,Y 297.531,Z 1128.874,A -85,B 0,C 180,E1 24334.817,E2 24334.817} C_VEL
LIN {X 0,Y 262.165,Z 1167.651,A -85,B 0,C 180,E1 24348.39,E2 24348.39} C_VEL
LIN {X 0,Y 240.594,Z 1192.044,A -85,B 0,C 180,E1 24365.905,E2 24365.905} C_VEL
LIN {X 0,Y 235.217,Z 1201.154,A -85,B 0,C 180,E1 24380.819,E2 24380.819} C_VEL
LIN {X 0,Y 235.153,Z 1202.612,A -85,B 0,C 180,E1 24391.947,E2 24391.947} C_VEL
LIN {X 0,Y 237.579,Z 1196.379,A -85,B 0,C 180,E1 24408.725,E2 24408.725} C_VEL
LIN {X 0,Y 254.226,Z 1176.15,A -85,B 0,C 180,E1 24426.94,E2 24426.94} C_VEL
LIN {X 0,Y 285.449,Z 1142.508,A -85,B 0,C 180,E1 24441.418,E2 24441.418} C_VEL
LIN {X 0,Y 323.828,Z 1096.525,A -85,B 0,C 180,E1 24451.711,E2 24451.711} C_VEL
LIN {X 0,Y 362.164,Z 1039.002,A -85,B 0,C 180,E1 24458.783,E2 24458.783} C_VEL
LIN {X 0,Y 384.099,Z 996.35,A -85,B 0,C 180,E1 24462.104,E2 24462.104} C_VEL
LIN {X 0,Y 380.262,Z 971.575,A -85,B 0,C 180,E1 24471.327,E2 24471.327} C_VEL
LIN {X 0,Y 378.992,Z 960,A -85,B 0,C 180,E1 24481.08,E2 24481.08} C_VEL
LIN {X 0,Y 378.902,Z 967.318,A -85,B 0,C 180,E1 24490.313,E2 24490.313} C_VEL
LIN {X 0,Y 379.94,Z 984.677,A -85,B 0,C 180,E1 24498.214,E2 24498.214} C_VEL
LIN {X 0,Y 378.254,Z 990.637,A -85,B 0,C 180,E1 24499.309,E2 24499.309} C_VEL
LIN {X 0,Y 360.054,Z 1022.968,A -85,B 0,C 180,E1 24501.978,E2 24501.978} C_VEL
LIN {X 0,Y 339.634,Z 1050.14,A -85,B 0,C 180,E1 24503.666,E2 24503.666} C_VEL
LIN {X 0,Y 297.654,Z 1103.95,A -85,B 0,C 180,E1 24512.599,E2 24512.599} C_VEL
LIN {X 0,Y 260.371,Z 1145.235,A -85,B 0,C 180,E1 24525.504,E2 24525.504} C_VEL
LIN {X 0,Y 236.135,Z 1172.431,A -85,B 0,C 180,E1 24542.123,E2 24542.123} C_VEL
LIN {X 0,Y 228.344,Z 1184.076,A -85,B 0,C 180,E1 24556.447,E2 24556.447} C_VEL
LIN {X 0,Y 227.316,Z 1187.398,A -85,B 0,C 180,E1 24571.811,E2 24571.811} C_VEL
LIN {X 0,Y 229.644,Z 1181.823,A -85,B 0,C 180,E1 24587.192,E2 24587.192} C_VEL
LIN {X 0,Y 244.112,Z 1162.957,A -85,B 0,C 180,E1 24604.981,E2 24604.981} C_VEL
LIN {X 0,Y 270.009,Z 1134.139,A -85,B 0,C 180,E1 24618.911,E2 24618.911} C_VEL
LIN {X 0,Y 237.386,Z 1130.525,A -85,B 0,C 180,E1 24635.571,E2 24635.571} C_VEL
LIN {X 0,Y 240.073,Z 1120.374,A -85,B 0,C 180,E1 24655.575,E2 24655.575} C_VEL
LIN {X 0,Y 267.624,Z 1104.498,A -85,B 0,C 180,E1 24667.827,E2 24667.827} C_VEL
LIN {X 0,Y 308.351,Z 1079.183,A -85,B 0,C 180,E1 24675.115,E2 24675.115} C_VEL
LIN {X 0,Y 352.814,Z 1042.568,A -85,B 0,C 180,E1 24679.038,E2 24679.038} C_VEL
LIN {X 0,Y 360.914,Z 1035.241,A -85,B 0,C 180,E1 24679.738,E2 24679.738} C_VEL
LIN {X 0,Y 322.36,Z 1092.516,A -85,B 0,C 180,E1 24686.418,E2 24686.418} C_VEL
LIN {X 0,Y 282.967,Z 1139.073,A -85,B 0,C 180,E1 24696.383,E2 24696.383} C_VEL
LIN {X 0,Y 249.807,Z 1173.4,A -85,B 0,C 180,E1 24710.494,E2 24710.494} C_VEL
LIN {X 0,Y 230.646,Z 1194.817,A -85,B 0,C 180,E1 24728.895,E2 24728.895} C_VEL
LIN {X 0,Y 227.071,Z 1201.869,A -85,B 0,C 180,E1 24744.35,E2 24744.35} C_VEL
LIN {X 0,Y 227.036,Z 1201.831,A -85,B 0,C 180,E1 24755.856,E2 24755.856} C_VEL
LIN {X 0,Y 230.758,Z 1194.664,A -85,B 0,C 180,E1 24771.309,E2 24771.309} C_VEL
LIN {X 0,Y 249.985,Z 1173.105,A -85,B 0,C 180,E1 24789.712,E2 24789.712} C_VEL
LIN {X 0,Y 284.36,Z 1137.563,A -85,B 0,C 180,E1 24804.096,E2 24804.096} C_VEL
LIN {X 0,Y 324.762,Z 1089.528,A -85,B 0,C 180,E1 24814.054,E2 24814.054} C_VEL
LIN {X 0,Y 364.001,Z 1029.883,A -85,B 0,C 180,E1 24820.774,E2 24820.774} C_VEL
LIN {X 0,Y 379.235,Z 1000.331,A -85,B 0,C 180,E1 24823.068,E2 24823.068} C_VEL
LIN {X 0,Y 376.21,Z 977.884,A -85,B 0,C 180,E1 24831.817,E2 24831.817} C_VEL
LIN {X 0,Y 375.351,Z 967.165,A -85,B 0,C 180,E1 24841.09,E2 24841.09} C_VEL
LIN {X 0,Y 374.987,Z 974.602,A -85,B 0,C 180,E1 24850.422,E2 24850.422} C_VEL
LIN {X 0,Y 375.304,Z 991.778,A -85,B 0,C 180,E1 24858.187,E2 24858.187} C_VEL
LIN {X 0,Y 339.634,Z 1050.14,A -85,B 0,C 180,E1 24863.666,E2 24863.666} C_VEL
LIN {X 0,Y 317.821,Z 1075.347,A -85,B 0,C 180,E1 24865.796,E2 24865.796} C_VEL
LIN {X 0,Y 276.329,Z 1122.863,A -85,B 0,C 180,E1 24875.997,E2 24875.997} C_VEL
LIN {X 0,Y 241.985,Z 1158.525,A -85,B 0,C 180,E1 24890.749,E2 24890.749} C_VEL
LIN {X 0,Y 223.936,Z 1179.169,A -85,B 0,C 180,E1 24908.009,E2 24908.009} C_VEL
LIN {X 0,Y 219.266,Z 1187.104,A -85,B 0,C 180,E1 24923.936,E2 24923.936} C_VEL
LIN {X 0,Y 219.324,Z 1187.128,A -85,B 0,C 180,E1 24935.851,E2 24935.851} C_VEL
LIN {X 0,Y 224.843,Z 1177.791,A -85,B 0,C 180,E1 24953.553,E2 24953.553} C_VEL
LIN {X 0,Y 245.59,Z 1154.571,A -85,B 0,C 180,E1 24971.318,E2 24971.318} C_VEL
LIN {X 0,Y 260.764,Z 1138.027,A -85,B 0,C 180,E1 24979.106,E2 24979.106} C_VEL
LIN {X 0,Y 228.38,Z 1133.403,A -85,B 0,C 180,E1 24998.688,E2 24998.688} C_VEL
LIN {X 0,Y 236.454,Z 1122.698,A -85,B 0,C 180,E1 25018.269,E2 25018.269} C_VEL
LIN {X 0,Y 266.503,Z 1106.967,A -85,B 0,C 180,E1 25029.747,E2 25029.747} C_VEL
LIN {X 0,Y 308.285,Z 1081.856,A -85,B 0,C 180,E1 25036.573,E2 25036.573} C_VEL
LIN {X 0,Y 347.044,Z 1052.39,A -85,B 0,C 180,E1 25040.14,E2 25040.14} C_VEL
LIN {X 0,Y 305.903,Z 1107.572,A -85,B 0,C 180,E1 25047.71,E2 25047.71} C_VEL
LIN {X 0,Y 264.622,Z 1152.087,A -85,B 0,C 180,E1 25059.415,E2 25059.415} C_VEL
LIN {X 0,Y 234.477,Z 1181.592,A -85,B 0,C 180,E1 25074.975,E2 25074.975} C_VEL
LIN {X 0,Y 220.457,Z 1198.297,A -85,B 0,C 180,E1 25094.35,E2 25094.35} C_VEL
LIN {X 0,Y 219.357,Z 1202.104,A -85,B 0,C 180,E1 25108.123,E2 25108.123} C_VEL
LIN {X 0,Y 220.003,Z 1199,A -85,B 0,C 180,E1 25124.077,E2 25124.077} C_VEL
LIN {X 0,Y 231.447,Z 1184.769,A -85,B 0,C 180,E1 25142.423,E2 25142.423} C_VEL
LIN {X 0,Y 261.14,Z 1155.653,A -85,B 0,C 180,E1 25159.191,E2 25159.191} C_VEL
LIN {X 0,Y 300.447,Z 1114.022,A -85,B 0,C 180,E1 25171.029,E2 25171.029} C_VEL
LIN {X 0,Y 342.186,Z 1059.808,A -85,B 0,C 180,E1 25179.106,E2 25179.106} C_VEL
LIN {X 0,Y 374.219,Z 1004.293,A -85,B 0,C 180,E1 25184.046,E2 25184.046} C_VEL
LIN {X 0,Y 371.957,Z 982.4,A -85,B 0,C 180,E1 25193.383,E2 25193.383} C_VEL
LIN {X 0,Y 371.621,Z 974.299,A -85,B 0,C 180,E1 25201.101,E2 25201.101} C_VEL
LIN {X 0,Y 370.907,Z 981.837,A -85,B 0,C 180,E1 25210.538,E2 25210.538} C_VEL
LIN {X 0,Y 370.125,Z 997.22,A -85,B 0,C 180,E1 25217.361,E2 25217.361} C_VEL
LIN {X 0,Y 331.419,Z 1057.572,A -85,B 0,C 180,E1 25223.254,E2 25223.254} C_VEL
LIN {X 0,Y 317.821,Z 1075.347,A -85,B 0,C 180,E1 25225.796,E2 25225.796} C_VEL
LIN {X 0,Y 294.946,Z 1098.427,A -85,B 0,C 180,E1 25228.472,E2 25228.472} C_VEL
LIN {X 0,Y 253.98,Z 1140.952,A -85,B 0,C 180,E1 25240.745,E2 25240.745} C_VEL
LIN {X 0,Y 223.78,Z 1170.927,A -85,B 0,C 180,E1 25258.208,E2 25258.208} C_VEL
LIN {X 0,Y 212.601,Z 1184.617,A -85,B 0,C 180,E1 25275.423,E2 25275.423} C_VEL
LIN {X 0,Y 211.311,Z 1187.925,A -85,B 0,C 180,E1 25291.948,E2 25291.948} C_VEL
LIN {X 0,Y 214.118,Z 1182.391,A -85,B 0,C 180,E1 25308.482,E2 25308.482} C_VEL
LIN {X 0,Y 230.695,Z 1163.596,A -85,B 0,C 180,E1 25327.347,E2 25327.347} C_VEL
LIN {X 0,Y 252.469,Z 1142.362,A -85,B 0,C 180,E1 25338.56,E2 25338.56} C_VEL
LIN {X 0,Y 220.338,Z 1136.032,A -85,B 0,C 180,E1 25362.07,E2 25362.07} C_VEL
LIN {X 0,Y 234.875,Z 1124.596,A -85,B 0,C 180,E1 25381.591,E2 25381.591} C_VEL
LIN {X 0,Y 267.79,Z 1108.36,A -85,B 0,C 180,E1 25392.084,E2 25392.084} C_VEL
LIN {X 0,Y 312.749,Z 1081.649,A -85,B 0,C 180,E1 25398.467,E2 25398.467} C_VEL
LIN {X 0,Y 333.64,Z 1066.866,A -85,B 0,C 180,E1 25400.44,E2 25400.44} C_VEL
LIN {X 0,Y 291.074,Z 1119.17,A -85,B 0,C 180,E1 25408.747,E2 25408.747} C_VEL
LIN {X 0,Y 251.079,Z 1159.316,A -85,B 0,C 180,E1 25421.079,E2 25421.079} C_VEL
LIN {X 0,Y 223.47,Z 1185.321,A -85,B 0,C 180,E1 25437.224,E2 25437.224} C_VEL
LIN {X 0,Y 212.107,Z 1198.81,A -85,B 0,C 180,E1 25455.612,E2 25455.612} C_VEL
LIN {X 0,Y 211.119,Z 1201.819,A -85,B 0,C 180,E1 25472.169,E2 25472.169} C_VEL
LIN {X 0,Y 214.381,Z 1195.481,A -85,B 0,C 180,E1 25490.84,E2 25490.84} C_VEL
LIN {X 0,Y 234.212,Z 1175.196,A -85,B 0,C 180,E1 25510.509,E2 25510.509} C_VEL
LIN {X 0,Y 270.551,Z 1140.717,A -85,B 0,C 180,E1 25525.698,E2 25525.698} C_VEL
LIN {X 0,Y 312.383,Z 1094.858,A -85,B 0,C 180,E1 25535.784,E2 25535.784} C_VEL
LIN {X 0,Y 354.635,Z 1035.396,A -85,B 0,C 180,E1 25542.721,E2 25542.721} C_VEL
LIN {X 0,Y 369.458,Z 1009.182,A -85,B 0,C 180,E1 25544.767,E2 25544.767} C_VEL
LIN {X 0,Y 367.754,Z 988.468,A -85,B 0,C 180,E1 25554.01,E2 25554.01} C_VEL
LIN {X 0,Y 367.695,Z 981.336,A -85,B 0,C 180,E1 25561.113,E2 25561.113} C_VEL
LIN {X 0,Y 366.746,Z 988.088,A -85,B 0,C 180,E1 25570.015,E2 25570.015} C_VEL
LIN {X 0,Y 365.444,Z 1001.884,A -85,B 0,C 180,E1 25576.446,E2 25576.446} C_VEL
LIN {X 0,Y 325.421,Z 1061.797,A -85,B 0,C 180,E1 25582.433,E2 25582.433} C_VEL
LIN {X 0,Y 294.946,Z 1098.427,A -85,B 0,C 180,E1 25588.472,E2 25588.472} C_VEL
LIN {X 0,Y 271.444,Z 1119.236,A -85,B 0,C 180,E1 25591.832,E2 25591.832} C_VEL
LIN {X 0,Y 232.107,Z 1156.452,A -85,B 0,C 180,E1 25606.517,E2 25606.517} C_VEL
LIN {X 0,Y 210.275,Z 1178.023,A -85,B 0,C 180,E1 25624.135,E2 25624.135} C_VEL
LIN {X 0,Y 203.284,Z 1187.636,A -85,B 0,C 180,E1 25643.457,E2 25643.457} C_VEL
LIN {X 0,Y 203.335,Z 1187.659,A -85,B 0,C 180,E1 25656.313,E2 25656.313} C_VEL
LIN {X 0,Y 208.623,Z 1179.829,A -85,B 0,C 180,E1 25673.459,E2 25673.459} C_VEL
LIN {X 0,Y 230.26,Z 1158.197,A -85,B 0,C 180,E1 25692.353,E2 25692.353} C_VEL
LIN {X 0,Y 243.094,Z 1145.504,A -85,B 0,C 180,E1 25699.193,E2 25699.193} C_VEL
LIN {X 0,Y 213.487,Z 1140.107,A -85,B 0,C 180,E1 25721.474,E2 25721.474} C_VEL
LIN {X 0,Y 228.153,Z 1129.056,A -85,B 0,C 180,E1 25742.017,E2 25742.017} C_VEL
LIN {X 0,Y 260.827,Z 1114.055,A -85,B 0,C 180,E1 25752.666,E2 25752.666} C_VEL
LIN {X 0,Y 308.872,Z 1087.097,A -85,B 0,C 180,E1 25759.496,E2 25759.496} C_VEL
LIN {X 0,Y 320.701,Z 1079.475,A -85,B 0,C 180,E1 25760.685,E2 25760.685} C_VEL
LIN {X 0,Y 277.213,Z 1128.86,A -85,B 0,C 180,E1 25769.68,E2 25769.68} C_VEL
LIN {X 0,Y 237.87,Z 1165.851,A -85,B 0,C 180,E1 25782.956,E2 25782.956} C_VEL
LIN {X 0,Y 210.742,Z 1190.728,A -85,B 0,C 180,E1 25802.219,E2 25802.219} C_VEL
LIN {X 0,Y 203.335,Z 1200.053,A -85,B 0,C 180,E1 25819.364,E2 25819.364} C_VEL
LIN {X 0,Y 203.128,Z 1201.557,A -85,B 0,C 180,E1 25832.254,E2 25832.254} C_VEL
LIN {X 0,Y 206.714,Z 1195.179,A -85,B 0,C 180,E1 25851.652,E2 25851.652} C_VEL
LIN {X 0,Y 227.853,Z 1174.805,A -85,B 0,C 180,E1 25871.889,E2 25871.889} C_VEL
LIN {X 0,Y 264.858,Z 1141.208,A -85,B 0,C 180,E1 25886.914,E2 25886.914} C_VEL
LIN {X 0,Y 309.015,Z 1094.22,A -85,B 0,C 180,E1 25897.216,E2 25897.216} C_VEL
LIN {X 0,Y 351.959,Z 1035.136,A -85,B 0,C 180,E1 25903.98,E2 25903.98} C_VEL
LIN {X 0,Y 364.526,Z 1013.255,A -85,B 0,C 180,E1 25905.744,E2 25905.744} C_VEL
LIN {X 0,Y 363.556,Z 993.908,A -85,B 0,C 180,E1 25915.142,E2 25915.142} C_VEL
LIN {X 0,Y 363.694,Z 988.314,A -85,B 0,C 180,E1 25921.125,E2 25921.125} C_VEL
LIN {X 0,Y 362.379,Z 994.777,A -85,B 0,C 180,E1 25929.906,E2 25929.906} C_VEL
LIN {X 0,Y 361.137,Z 1006.058,A -85,B 0,C 180,E1 25935.472,E2 25935.472} C_VEL
LIN {X 0,Y 318.044,Z 1067.78,A -85,B 0,C 180,E1 25941.814,E2 25941.814} C_VEL
LIN {X 0,Y 271.444,Z 1119.236,A -85,B 0,C 180,E1 25951.832,E2 25951.832} C_VEL
LIN {X 0,Y 248.102,Z 1137.589,A -85,B 0,C 180,E1 25956.13,E2 25956.13} C_VEL
LIN {X 0,Y 212.686,Z 1169.047,A -85,B 0,C 180,E1 25973.693,E2 25973.693} C_VEL
LIN {X 0,Y 196.922,Z 1185.16,A -85,B 0,C 180,E1 25994.233,E2 25994.233} C_VEL
LIN {X 0,Y 195.3,Z 1188.453,A -85,B 0,C 180,E1 26012.108,E2 26012.108} C_VEL
LIN {X 0,Y 198.705,Z 1182.962,A -85,B 0,C 180,E1 26029.974,E2 26029.974} C_VEL
LIN {X 0,Y 217.545,Z 1164.405,A -85,B 0,C 180,E1 26049.891,E2 26049.891} C_VEL
LIN {X 0,Y 234.303,Z 1148.81,A -85,B 0,C 180,E1 26059.298,E2 26059.298} C_VEL
LIN {X 0,Y 206.583,Z 1144.061,A -85,B 0,C 180,E1 26080.831,E2 26080.831} C_VEL
LIN {X 0,Y 220.688,Z 1133.733,A -85,B 0,C 180,E1 26102.086,E2 26102.086} C_VEL
LIN {X 0,Y 254.745,Z 1119.043,A -85,B 0,C 180,E1 26113.487,E2 26113.487} C_VEL
LIN {X 0,Y 303.134,Z 1093.593,A -85,B 0,C 180,E1 26120.374,E2 26120.374} C_VEL
LIN {X 0,Y 308.061,Z 1090.541,A -85,B 0,C 180,E1 26120.828,E2 26120.828} C_VEL
LIN {X 0,Y 262.25,Z 1138.866,A -85,B 0,C 180,E1 26131.044,E2 26131.044} C_VEL
LIN {X 0,Y 222.556,Z 1173.724,A -85,B 0,C 180,E1 26146.288,E2 26146.288} C_VEL
LIN {X 0,Y 198.969,Z 1194.983,A -85,B 0,C 180,E1 26167.711,E2 26167.711} C_VEL
LIN {X 0,Y 195.291,Z 1201.311,A -85,B 0,C 180,E1 26187.892,E2 26187.892} C_VEL
LIN {X 0,Y 196.386,Z 1198.15,A -85,B 0,C 180,E1 26205.811,E2 26205.811} C_VEL
LIN {X 0,Y 211.332,Z 1183.255,A -85,B 0,C 180,E1 26226.459,E2 26226.459} C_VEL
LIN {X 0,Y 246.666,Z 1153.087,A -85,B 0,C 180,E1 26244.116,E2 26244.116} C_VEL
LIN {X 0,Y 290.147,Z 1111.005,A -85,B 0,C 180,E1 26255.671,E2 26255.671} C_VEL
LIN {X 0,Y 334.829,Z 1056.52,A -85,B 0,C 180,E1 26263.282,E2 26263.282} C_VEL
LIN {X 0,Y 359.65,Z 1018.062,A -85,B 0,C 180,E1 26266.511,E2 26266.511} C_VEL
LIN {X 0,Y 359.179,Z 1000.824,A -85,B 0,C 180,E1 26275.082,E2 26275.082} C_VEL
LIN {X 0,Y 359.505,Z 995.183,A -85,B 0,C 180,E1 26281.138,E2 26281.138} C_VEL
LIN {X 0,Y 358.003,Z 1001.838,A -85,B 0,C 180,E1 26290.029,E2 26290.029} C_VEL
LIN {X 0,Y 356.002,Z 1011.504,A -85,B 0,C 180,E1 26294.586,E2 26294.586} C_VEL
LIN {X 0,Y 312.561,Z 1071.329,A -85,B 0,C 180,E1 26300.853,E2 26300.853} C_VEL
LIN {X 0,Y 265.345,Z 1121.469,A -85,B 0,C 180,E1 26310.82,E2 26310.82} C_VEL
LIN {X 0,Y 248.102,Z 1137.589,A -85,B 0,C 180,E1 26316.13,E2 26316.13} C_VEL
LIN {X 0,Y 224.978,Z 1153.425,A -85,B 0,C 180,E1 26321.43,E2 26321.43} C_VEL
LIN {X 0,Y 197.329,Z 1176.914,A -85,B 0,C 180,E1 26339.878,E2 26339.878} C_VEL
LIN {X 0,Y 187.876,Z 1187.077,A -85,B 0,C 180,E1 26358.226,E2 26358.226} C_VEL
LIN {X 0,Y 187.319,Z 1188.716,A -85,B 0,C 180,E1 26372.198,E2 26372.198} C_VEL
LIN {X 0,Y 191.039,Z 1183.248,A -85,B 0,C 180,E1 26390.812,E2 26390.812} C_VEL
LIN {X 0,Y 210.944,Z 1165,A -85,B 0,C 180,E1 26411.139,E2 26411.139} C_VEL
LIN {X 0,Y 225.44,Z 1152.097,A -85,B 0,C 180,E1 26419.444,E2 26419.444} C_VEL
LIN {X 0,Y 199.163,Z 1146.427,A -85,B 0,C 180,E1 26444.669,E2 26444.669} C_VEL
LIN {X 0,Y 216.842,Z 1136.715,A -85,B 0,C 180,E1 26464.132,E2 26464.132} C_VEL
LIN {X 0,Y 255.157,Z 1121.079,A -85,B 0,C 180,E1 26475.624,E2 26475.624} C_VEL
LIN {X 0,Y 294.888,Z 1101.288,A -85,B 0,C 180,E1 26481.055,E2 26481.055} C_VEL
LIN {X 0,Y 248.745,Z 1146.488,A -85,B 0,C 180,E1 26491.996,E2 26491.996} C_VEL
LIN {X 0,Y 208.894,Z 1179.38,A -85,B 0,C 180,E1 26509.099,E2 26509.099} C_VEL
LIN {X 0,Y 189.247,Z 1197.028,A -85,B 0,C 180,E1 26531.423,E2 26531.423} C_VEL
LIN {X 0,Y 187.271,Z 1201.046,A -85,B 0,C 180,E1 26547.802,E2 26547.802} C_VEL
LIN {X 0,Y 188.544,Z 1197.868,A -85,B 0,C 180,E1 26566.487,E2 26566.487} C_VEL
LIN {X 0,Y 206.146,Z 1181.736,A -85,B 0,C 180,E1 26588.873,E2 26588.873} C_VEL
LIN {X 0,Y 243.464,Z 1151.174,A -85,B 0,C 180,E1 26606.298,E2 26606.298} C_VEL
LIN {X 0,Y 288.955,Z 1108.061,A -85,B 0,C 180,E1 26617.642,E2 26617.642} C_VEL
LIN {X 0,Y 334.36,Z 1053.173,A -85,B 0,C 180,E1 26624.913,E2 26624.913} C_VEL
LIN {X 0,Y 354.65,Z 1022.127,A -85,B 0,C 180,E1 26627.578,E2 26627.578} C_VEL
LIN {X 0,Y 354.838,Z 1006.281,A -85,B 0,C 180,E1 26636.251,E2 26636.251} C_VEL
LIN {X 0,Y 354.812,Z 1002.265,A -85,B 0,C 180,E1 26643.606,E2 26643.606} C_VEL
LIN {X 0,Y 352.733,Z 1013.023,A -85,B 0,C 180,E1 26652.712,E2 26652.712} C_VEL
LIN {X 0,Y 349.194,Z 1019.546,A -85,B 0,C 180,E1 26653.893,E2 26653.893} C_VEL
LIN {X 0,Y 304.109,Z 1078.18,A -85,B 0,C 180,E1 26660.361,E2 26660.361} C_VEL
LIN {X 0,Y 256.059,Z 1126.477,A -85,B 0,C 180,E1 26670.593,E2 26670.593} C_VEL
LIN {X 0,Y 224.978,Z 1153.425,A -85,B 0,C 180,E1 26681.43,E2 26681.43} C_VEL
LIN {X 0,Y 203.478,Z 1166.517,A -85,B 0,C 180,E1 26688.136,E2 26688.136} C_VEL
LIN {X 0,Y 182.301,Z 1184.585,A -85,B 0,C 180,E1 26710.419,E2 26710.419} C_VEL
LIN {X 0,Y 179.106,Z 1188.978,A -85,B 0,C 180,E1 26727.443,E2 26727.443} C_VEL
LIN {X 0,Y 181.042,Z 1186.096,A -85,B 0,C 180,E1 26745.988,E2 26745.988} C_VEL
LIN {X 0,Y 197.644,Z 1171.15,A -85,B 0,C 180,E1 26767.744,E2 26767.744} C_VEL
LIN {X 0,Y 216.318,Z 1155.27,A -85,B 0,C 180,E1 26779.704,E2 26779.704} C_VEL
LIN {X 0,Y 191.952,Z 1150.125,A -85,B 0,C 180,E1 26804.078,E2 26804.078} C_VEL
LIN {X 0,Y 213.308,Z 1139.586,A -85,B 0,C 180,E1 26826.245,E2 26826.245} C_VEL
LIN {X 0,Y 252.779,Z 1124.383,A -85,B 0,C 180,E1 26837.207,E2 26837.207} C_VEL
LIN {X 0,Y 282.182,Z 1110.816,A -85,B 0,C 180,E1 26841.282,E2 26841.282} C_VEL
LIN {X 0,Y 234.708,Z 1153.998,A -85,B 0,C 180,E1 26853.279,E2 26853.279} C_VEL
LIN {X 0,Y 197.605,Z 1182.748,A -85,B 0,C 180,E1 26870.843,E2 26870.843} C_VEL
LIN {X 0,Y 180.668,Z 1197.676,A -85,B 0,C 180,E1 26893.039,E2 26893.039} C_VEL
LIN {X 0,Y 179.246,Z 1200.782,A -85,B 0,C 180,E1 26907.703,E2 26907.703} C_VEL
LIN {X 0,Y 180.746,Z 1197.576,A -85,B 0,C 180,E1 26927.22,E2 26927.22} C_VEL
LIN {X 0,Y 199.714,Z 1181.353,A -85,B 0,C 180,E1 26950.376,E2 26950.376} C_VEL
LIN {X 0,Y 238.775,Z 1150.703,A -85,B 0,C 180,E1 26967.99,E2 26967.99} C_VEL
LIN {X 0,Y 286.201,Z 1107.07,A -85,B 0,C 180,E1 26979.286,E2 26979.286} C_VEL
LIN {X 0,Y 332.262,Z 1052.469,A -85,B 0,C 180,E1 26986.32,E2 26986.32} C_VEL
LIN {X 0,Y 349.724,Z 1026.308,A -85,B 0,C 180,E1 26988.668,E2 26988.668} C_VEL
LIN {X 0,Y 350.245,Z 1011.722,A -85,B 0,C 180,E1 26997.444,E2 26997.444} C_VEL
LIN {X 0,Y 350.459,Z 1009.076,A -85,B 0,C 180,E1 27003.651,E2 27003.651} C_VEL
LIN {X 0,Y 347.852,Z 1019.138,A -85,B 0,C 180,E1 27012.437,E2 27012.437} C_VEL
LIN {X 0,Y 301.699,Z 1078.314,A -85,B 0,C 180,E1 27018.836,E2 27018.836} C_VEL
LIN {X 0,Y 251.93,Z 1126.879,A -85,B 0,C 180,E1 27028.966,E2 27028.966} C_VEL
LIN {X 0,Y 208.999,Z 1162.059,A -85,B 0,C 180,E1 27044.828,E2 27044.828} C_VEL
LIN {X 0,Y 203.478,Z 1166.517,A -85,B 0,C 180,E1 27048.136,E2 27048.136} C_VEL
LIN {X 0,Y 184.138,Z 1176.854,A -85,B 0,C 180,E1 27056.45,E2 27056.45} C_VEL
LIN {X 0,Y 172.051,Z 1187.612,A -85,B 0,C 180,E1 27077.125,E2 27077.125} C_VEL
LIN {X 0,Y 171.295,Z 1189.244,A -85,B 0,C 180,E1 27092.404,E2 27092.404} C_VEL
LIN {X 0,Y 175.852,Z 1183.823,A -85,B 0,C 180,E1 27112.705,E2 27112.705} C_VEL
LIN {X 0,Y 198.562,Z 1165.785,A -85,B 0,C 180,E1 27134.2,E2 27134.2} C_VEL
LIN {X 0,Y 207.709,Z 1158.279,A -85,B 0,C 180,E1 27139.725,E2 27139.725} C_VEL
LIN {X 0,Y 185.453,Z 1152.348,A -85,B 0,C 180,E1 27168.338,E2 27168.338} C_VEL
LIN {X 0,Y 210.183,Z 1142.348,A -85,B 0,C 180,E1 27188.478,E2 27188.478} C_VEL
LIN {X 0,Y 253.681,Z 1126.369,A -85,B 0,C 180,E1 27199.312,E2 27199.312} C_VEL
LIN {X 0,Y 269.099,Z 1120.181,A -85,B 0,C 180,E1 27201.741,E2 27201.741} C_VEL
LIN {X 0,Y 220.785,Z 1160.692,A -85,B 0,C 180,E1 27214.627,E2 27214.627} C_VEL
LIN {X 0,Y 185.16,Z 1186.902,A -85,B 0,C 180,E1 27234.067,E2 27234.067} C_VEL
LIN {X 0,Y 171.567,Z 1198.954,A -85,B 0,C 180,E1 27257.364,E2 27257.364} C_VEL
LIN {X 0,Y 171.07,Z 1200.498,A -85,B 0,C 180,E1 27272.677,E2 27272.677} C_VEL
LIN {X 0,Y 176.005,Z 1194.34,A -85,B 0,C 180,E1 27294.813,E2 27294.813} C_VEL
LIN {X 0,Y 203.608,Z 1173.484,A -85,B 0,C 180,E1 27318.039,E2 27318.039} C_VEL
LIN {X 0,Y 249.209,Z 1138.026,A -85,B 0,C 180,E1 27333.849,E2 27333.849} C_VEL
LIN {X 0,Y 300.376,Z 1088.496,A -85,B 0,C 180,E1 27343.687,E2 27343.687} C_VEL
LIN {X 0,Y 344.734,Z 1031.029,A -85,B 0,C 180,E1 27349.506,E2 27349.506} C_VEL
LIN {X 0,Y 345.682,Z 1018.757,A -85,B 0,C 180,E1 27357.093,E2 27357.093} C_VEL
LIN {X 0,Y 345.742,Z 1015.661,A -85,B 0,C 180,E1 27363.7,E2 27363.7} C_VEL
LIN {X 0,Y 342.618,Z 1025.174,A -85,B 0,C 180,E1 27371.62,E2 27371.62} C_VEL
LIN {X 0,Y 293.893,Z 1084.534,A -85,B 0,C 180,E1 27378.186,E2 27378.186} C_VEL
LIN {X 0,Y 242.649,Z 1131.864,A -85,B 0,C 180,E1 27388.704,E2 27388.704} C_VEL
LIN {X 0,Y 198.729,Z 1165.773,A -85,B 0,C 180,E1 27405.666,E2 27405.666} C_VEL
LIN {X 0,Y 184.138,Z 1176.854,A -85,B 0,C 180,E1 27416.45,E2 27416.45} C_VEL
LIN {X 0,Y 168.118,Z 1184.296,A -85,B 0,C 180,E1 27426.509,E2 27426.509} C_VEL
LIN {X 0,Y 163.106,Z 1189.506,A -85,B 0,C 180,E1 27447.192,E2 27447.192} C_VEL
LIN {X 0,Y 164.678,Z 1187.319,A -85,B 0,C 180,E1 27465.267,E2 27465.267} C_VEL
LIN {X 0,Y 181.78,Z 1173.949,A -85,B 0,C 180,E1 27488.595,E2 27488.595} C_VEL
LIN {X 0,Y 199.012,Z 1161.252,A -85,B 0,C 180,E1 27499.774,E2 27499.774} C_VEL
LIN {X 0,Y 178.043,Z 1155.869,A -85,B 0,C 180,E1 27527.905,E2 27527.905} C_VEL
LIN {X 0,Y 203.282,Z 1146.369,A -85,B 0,C 180,E1 27549.171,E2 27549.171} C_VEL
LIN {X 0,Y 247.347,Z 1131.234,A -85,B 0,C 180,E1 27560.276,E2 27560.276} C_VEL
LIN {X 0,Y 256.489,Z 1127.681,A -85,B 0,C 180,E1 27561.608,E2 27561.608} C_VEL
LIN {X 0,Y 211.295,Z 1163.662,A -85,B 0,C 180,E1 27574.521,E2 27574.521} C_VEL
LIN {X 0,Y 175.164,Z 1188.933,A -85,B 0,C 180,E1 27595.631,E2 27595.631} C_VEL
LIN {X 0,Y 163.46,Z 1198.934,A -85,B 0,C 180,E1 27617.78,E2 27617.78} C_VEL
LIN {X 0,Y 163.048,Z 1200.235,A -85,B 0,C 180,E1 27632.809,E2 27632.809} C_VEL
LIN {X 0,Y 168.531,Z 1194.031,A -85,B 0,C 180,E1 27655.994,E2 27655.994} C_VEL
LIN {X 0,Y 196.866,Z 1173.882,A -85,B 0,C 180,E1 27679.256,E2 27679.256} C_VEL
LIN {X 0,Y 243.134,Z 1139.439,A -85,B 0,C 180,E1 27695.034,E2 27695.034} C_VEL
LIN {X 0,Y 293.484,Z 1092.678,A -85,B 0,C 180,E1 27704.568,E2 27704.568} C_VEL
LIN {X 0,Y 339.848,Z 1035.329,A -85,B 0,C 180,E1 27710.584,E2 27710.584} C_VEL
LIN {X 0,Y 341.021,Z 1023.839,A -85,B 0,C 180,E1 27718.651,E2 27718.651} C_VEL
LIN {X 0,Y 341.117,Z 1022.313,A -85,B 0,C 180,E1 27723.751,E2 27723.751} C_VEL
LIN {X 0,Y 337.599,Z 1030.533,A -85,B 0,C 180,E1 27730.66,E2 27730.66} C_VEL
LIN {X 0,Y 289.419,Z 1087.027,A -85,B 0,C 180,E1 27736.961,E2 27736.961} C_VEL
LIN {X 0,Y 237.37,Z 1133.401,A -85,B 0,C 180,E1 27747.323,E2 27747.323} C_VEL
LIN {X 0,Y 193.156,Z 1165.914,A -85,B 0,C 180,E1 27763.787,E2 27763.787} C_VEL
LIN {X 0,Y 168.118,Z 1184.296,A -85,B 0,C 180,E1 27786.509,E2 27786.509} C_VEL
LIN {X 0,Y 155.733,Z 1188.617,A -85,B 0,C 180,E1 27798.193,E2 27798.193} C_VEL
LIN {X 0,Y 155.268,Z 1189.771,A -85,B 0,C 180,E1 27812.652,E2 27812.652} C_VEL
LIN {X 0,Y 160.876,Z 1184.4,A -85,B 0,C 180,E1 27834.956,E2 27834.956} C_VEL
LIN {X 0,Y 187.824,Z 1165.919,A -85,B 0,C 180,E1 27858.17,E2 27858.17} C_VEL
LIN {X 0,Y 189.865,Z 1164.566,A -85,B 0,C 180,E1 27859.208,E2 27859.208} C_VEL
LIN {X 0,Y 176.518,Z 1156.308,A -85,B 0,C 180,E1 27897.681,E2 27897.681} C_VEL
LIN {X 0,Y 217.217,Z 1143.969,A -85,B 0,C 180,E1 27916.624,E2 27916.624} C_VEL
LIN {X 0,Y 244.801,Z 1134.607,A -85,B 0,C 180,E1 27921.86,E2 27921.86} C_VEL
LIN {X 0,Y 197.209,Z 1169.661,A -85,B 0,C 180,E1 27936.309,E2 27936.309} C_VEL
LIN {X 0,Y 163.519,Z 1192.009,A -85,B 0,C 180,E1 27959.476,E2 27959.476} C_VEL
LIN {X 0,Y 155.048,Z 1199.456,A -85,B 0,C 180,E1 27981.709,E2 27981.709} C_VEL
LIN {X 0,Y 155.044,Z 1199.413,A -85,B 0,C 180,E1 27998.592,E2 27998.592} C_VEL
LIN {X 0,Y 165.67,Z 1190.468,A -85,B 0,C 180,E1 28023.247,E2 28023.247} C_VEL
LIN {X 0,Y 201.579,Z 1166.815,A -85,B 0,C 180,E1 28045.478,E2 28045.478} C_VEL
LIN {X 0,Y 251.65,Z 1129.242,A -85,B 0,C 180,E1 28059.42,E2 28059.42} C_VEL
LIN {X 0,Y 303.179,Z 1079.3,A -85,B 0,C 180,E1 28067.756,E2 28067.756} C_VEL
LIN {X 0,Y 334.907,Z 1039.647,A -85,B 0,C 180,E1 28071.69,E2 28071.69} C_VEL
LIN {X 0,Y 336.194,Z 1030.336,A -85,B 0,C 180,E1 28078.631,E2 28078.631} C_VEL
LIN {X 0,Y 336.138,Z 1028.729,A -85,B 0,C 180,E1 28083.806,E2 28083.806} C_VEL
LIN {X 0,Y 333.183,Z 1035.072,A -85,B 0,C 180,E1 28089.612,E2 28089.612} C_VEL
LIN {X 0,Y 283.282,Z 1091.193,A -85,B 0,C 180,E1 28095.97,E2 28095.97} C_VEL
LIN {X 0,Y 231.8,Z 1135.202,A -85,B 0,C 180,E1 28105.993,E2 28105.993} C_VEL
LIN {X 0,Y 184.294,Z 1168.415,A -85,B 0,C 180,E1 28123.734,E2 28123.734} C_VEL
LIN {X 0,Y 159.481,Z 1185.438,A -85,B 0,C 180,E1 28147.475,E2 28147.475} C_VEL
LIN {X 0,Y 155.733,Z 1188.617,A -85,B 0,C 180,E1 28158.193,E2 28158.193} C_VEL
LIN {X 0,Y 147.064,Z 1190.035,A -85,B 0,C 180,E1 28171.316,E2 28171.316} C_VEL
LIN {X 0,Y 153.509,Z 1184.687,A -85,B 0,C 180,E1 28196.243,E2 28196.243} C_VEL
LIN {X 0,Y 179.11,Z 1168.383,A -85,B 0,C 180,E1 28218.405,E2 28218.405} C_VEL
LIN {X 0,Y 179.61,Z 1166.643,A -85,B 0,C 180,E1 28220.87,E2 28220.87} C_VEL
LIN {X 0,Y 168.757,Z 1159.722,A -85,B 0,C 180,E1 28257.575,E2 28257.575} C_VEL
LIN {X 0,Y 210.319,Z 1148.133,A -85,B 0,C 180,E1 28277.52,E2 28277.52} C_VEL
LIN {X 0,Y 231.836,Z 1141.993,A -85,B 0,C 180,E1 28282.373,E2 28282.373} C_VEL
LIN {X 0,Y 182.455,Z 1175.562,A -85,B 0,C 180,E1 28298.764,E2 28298.764} C_VEL
LIN {X 0,Y 152.518,Z 1194.392,A -85,B 0,C 180,E1 28323.574,E2 28323.574} C_VEL
LIN {X 0,Y 147.156,Z 1199.724,A -85,B 0,C 180,E1 28347.202,E2 28347.202} C_VEL
LIN {X 0,Y 147.923,Z 1198.06,A -85,B 0,C 180,E1 28365.02,E2 28365.02} C_VEL
LIN {X 0,Y 166.393,Z 1185.457,A -85,B 0,C 180,E1 28391.571,E2 28391.571} C_VEL
LIN {X 0,Y 210.325,Z 1157.579,A -85,B 0,C 180,E1 28411.9,E2 28411.9} C_VEL
LIN {X 0,Y 264.395,Z 1115.451,A -85,B 0,C 180,E1 28424.011,E2 28424.011} C_VEL
LIN {X 0,Y 316.516,Z 1061.563,A -85,B 0,C 180,E1 28431.051,E2 28431.051} C_VEL
LIN {X 0,Y 329.493,Z 1045.065,A -85,B 0,C 180,E1 28432.441,E2 28432.441} C_VEL
LIN {X 0,Y 331.189,Z 1036.685,A -85,B 0,C 180,E1 28438.61,E2 28438.61} C_VEL
LIN {X 0,Y 331.246,Z 1035.212,A -85,B 0,C 180,E1 28443.863,E2 28443.863} C_VEL
LIN {X 0,Y 328.341,Z 1040.31,A -85,B 0,C 180,E1 28448.596,E2 28448.596} C_VEL
LIN {X 0,Y 276.789,Z 1095.834,A -85,B 0,C 180,E1 28455.002,E2 28455.002} C_VEL
LIN {X 0,Y 221.692,Z 1140.374,A -85,B 0,C 180,E1 28465.807,E2 28465.807} C_VEL
LIN {X 0,Y 174.689,Z 1171.169,A -85,B 0,C 180,E1 28484.119,E2 28484.119} C_VEL
LIN {X 0,Y 150.565,Z 1186.802,A -85,B 0,C 180,E1 28509.183,E2 28509.183} C_VEL
LIN {X 0,Y 147.064,Z 1190.035,A -85,B 0,C 180,E1 28531.316,E2 28531.316} C_VEL
LIN {X 0,Y 140.561,Z 1188.769,A -85,B 0,C 180,E1 28545.302,E2 28545.302} C_VEL
LIN {X 0,Y 160.697,Z 1176.262,A -85,B 0,C 180,E1 28572.403,E2 28572.403} C_VEL
LIN {X 0,Y 171.534,Z 1169.23,A -85,B 0,C 180,E1 28580.653,E2 28580.653} C_VEL
LIN {X 0,Y 160.996,Z 1163.053,A -85,B 0,C 180,E1 28617.458,E2 28617.458} C_VEL
LIN {X 0,Y 202.364,Z 1152.368,A -85,B 0,C 180,E1 28638.227,E2 28638.227} C_VEL
LIN {X 0,Y 220.081,Z 1147.712,A -85,B 0,C 180,E1 28642.408,E2 28642.408} C_VEL
LIN {X 0,Y 171.193,Z 1178.723,A -85,B 0,C 180,E1 28659.664,E2 28659.664} C_VEL
LIN {X 0,Y 144.185,Z 1194.804,A -85,B 0,C 180,E1 28683.836,E2 28683.836} C_VEL
LIN {X 0,Y 139.139,Z 1199.458,A -85,B 0,C 180,E1 28707.04,E2 28707.04} C_VEL
LIN {X 0,Y 140.069,Z 1197.783,A -85,B 0,C 180,E1 28725.884,E2 28725.884} C_VEL
LIN {X 0,Y 160.246,Z 1185.126,A -85,B 0,C 180,E1 28753.551,E2 28753.551} C_VEL
LIN {X 0,Y 205.833,Z 1157.593,A -85,B 0,C 180,E1 28773.777,E2 28773.777} C_VEL
LIN {X 0,Y 261.933,Z 1115.125,A -85,B 0,C 180,E1 28785.768,E2 28785.768} C_VEL
LIN {X 0,Y 315.838,Z 1060.267,A -85,B 0,C 180,E1 28792.617,E2 28792.617} C_VEL
LIN {X 0,Y 324.977,Z 1048.606,A -85,B 0,C 180,E1 28793.824,E2 28793.824} C_VEL
LIN {X 0,Y 326.73,Z 1040.979,A -85,B 0,C 180,E1 28801.417,E2 28801.417} C_VEL
LIN {X 0,Y 323.569,Z 1045.441,A -85,B 0,C 180,E1 28807.561,E2 28807.561} C_VEL
LIN {X 0,Y 269.481,Z 1101.063,A -85,B 0,C 180,E1 28814.1,E2 28814.1} C_VEL
LIN {X 0,Y 212.942,Z 1144.369,A -85,B 0,C 180,E1 28825.226,E2 28825.226} C_VEL
LIN {X 0,Y 166.11,Z 1173.266,A -85,B 0,C 180,E1 28843.904,E2 28843.904} C_VEL
LIN {X 0,Y 142.974,Z 1187.079,A -85,B 0,C 180,E1 28868.021,E2 28868.021} C_VEL
LIN {X 0,Y 139.251,Z 1190.3,A -85,B 0,C 180,E1 28892.957,E2 28892.957} C_VEL
LIN {X 0,Y 140.561,Z 1188.769,A -85,B 0,C 180,E1 28905.302,E2 28905.302} C_VEL
LIN {X 0,Y 139.399,Z 1185,A -85,B 0,C 180,E1 28919.819,E2 28919.819} C_VEL
LIN {X 0,Y 162.751,Z 1172.154,A -85,B 0,C 180,E1 28939.641,E2 28939.641} C_VEL
LIN {X 0,Y 159.17,Z 1164.588,A -85,B 0,C 180,E1 28983.227,E2 28983.227} C_VEL
LIN {X 0,Y 208.13,Z 1152.932,A -85,B 0,C 180,E1 29002.18,E2 29002.18} C_VEL
LIN {X 0,Y 159.736,Z 1181.729,A -85,B 0,C 180,E1 29020.764,E2 29020.764} C_VEL
LIN {X 0,Y 134.474,Z 1195.966,A -85,B 0,C 180,E1 29046.925,E2 29046.925} C_VEL
LIN {X 0,Y 131.105,Z 1199.194,A -85,B 0,C 180,E1 29066.859,E2 29066.859} C_VEL
LIN {X 0,Y 132.245,Z 1197.504,A -85,B 0,C 180,E1 29086.851,E2 29086.851} C_VEL
LIN {X 0,Y 154.309,Z 1184.791,A -85,B 0,C 180,E1 29115.685,E2 29115.685} C_VEL
LIN {X 0,Y 202.44,Z 1157.011,A -85,B 0,C 180,E1 29135.999,E2 29135.999} C_VEL
LIN {X 0,Y 259.229,Z 1115.169,A -85,B 0,C 180,E1 29147.471,E2 29147.471} C_VEL
LIN {X 0,Y 313.187,Z 1061.479,A -85,B 0,C 180,E1 29153.973,E2 29153.973} C_VEL
LIN {X 0,Y 319.876,Z 1053.09,A -85,B 0,C 180,E1 29154.97,E2 29154.97} C_VEL
LIN {X 0,Y 321.574,Z 1047.123,A -85,B 0,C 180,E1 29161.272,E2 29161.272} C_VEL
LIN {X 0,Y 318.49,Z 1050.738,A -85,B 0,C 180,E1 29166.513,E2 29166.513} C_VEL
LIN {X 0,Y 264.497,Z 1104.152,A -85,B 0,C 180,E1 29172.812,E2 29172.812} C_VEL
LIN {X 0,Y 207.544,Z 1146.009,A -85,B 0,C 180,E1 29183.68,E2 29183.68} C_VEL
LIN {X 0,Y 157.584,Z 1175.12,A -85,B 0,C 180,E1 29203.555,E2 29203.555} C_VEL
LIN {X 0,Y 135.442,Z 1187.354,A -85,B 0,C 180,E1 29226.73,E2 29226.73} C_VEL
LIN {X 0,Y 131.091,Z 1190.563,A -85,B 0,C 180,E1 29246.506,E2 29246.506} C_VEL
LIN {X 0,Y 132.816,Z 1189.008,A -85,B 0,C 180,E1 29266.414,E2 29266.414} C_VEL
LIN {X 0,Y 139.399,Z 1185,A -85,B 0,C 180,E1 29279.819,E2 29279.819} C_VEL
LIN {X 0,Y 144.873,Z 1178.956,A -85,B 0,C 180,E1 29293.81,E2 29293.81} C_VEL
LIN {X 0,Y 154.627,Z 1173.884,A -85,B 0,C 180,E1 29300.586,E2 29300.586} C_VEL
LIN {X 0,Y 145.259,Z 1169.159,A -85,B 0,C 180,E1 29337.182,E2 29337.182} C_VEL
LIN {X 0,Y 184.299,Z 1160.69,A -85,B 0,C 180,E1 29359.159,E2 29359.159} C_VEL
LIN {X 0,Y 196.519,Z 1157.934,A -85,B 0,C 180,E1 29362.304,E2 29362.304} C_VEL
LIN {X 0,Y 148.666,Z 1184.275,A -85,B 0,C 180,E1 29381.787,E2 29381.787} C_VEL
LIN {X 0,Y 126.959,Z 1195.673,A -85,B 0,C 180,E1 29405.473,E2 29405.473} C_VEL
LIN {X 0,Y 123.092,Z 1198.93,A -85,B 0,C 180,E1 29426.654,E2 29426.654} C_VEL
LIN {X 0,Y 124.456,Z 1197.232,A -85,B 0,C 180,E1 29447.94,E2 29447.94} C_VEL
LIN {X 0,Y 149.314,Z 1184.085,A -85,B 0,C 180,E1 29478.435,E2 29478.435} C_VEL
LIN {X 0,Y 201.317,Z 1155.123,A -85,B 0,C 180,E1 29498.828,E2 29498.828} C_VEL
LIN {X 0,Y 259.14,Z 1113.304,A -85,B 0,C 180,E1 29509.526,E2 29509.526} C_VEL
LIN {X 0,Y 314.7,Z 1058.166,A -85,B 0,C 180,E1 29515.772,E2 29515.772} C_VEL
LIN {X 0,Y 316.316,Z 1053.2,A -85,B 0,C 180,E1 29521.294,E2 29521.294} C_VEL
LIN {X 0,Y 313.857,Z 1055.688,A -85,B 0,C 180,E1 29525.404,E2 29525.404} C_VEL
LIN {X 0,Y 259.092,Z 1107.702,A -85,B 0,C 180,E1 29531.561,E2 29531.561} C_VEL
LIN {X 0,Y 201.273,Z 1148.287,A -85,B 0,C 180,E1 29542.31,E2 29542.31} C_VEL
LIN {X 0,Y 151.983,Z 1175.45,A -85,B 0,C 180,E1 29561.287,E2 29561.287} C_VEL
LIN {X 0,Y 127.984,Z 1187.63,A -85,B 0,C 180,E1 29585.286,E2 29585.286} C_VEL
LIN {X 0,Y 123.095,Z 1190.826,A -85,B 0,C 180,E1 29606.279,E2 29606.279} C_VEL
LIN {X 0,Y 125.05,Z 1189.278,A -85,B 0,C 180,E1 29627.465,E2 29627.465} C_VEL
LIN {X 0,Y 144.873,Z 1178.956,A -85,B 0,C 180,E1 29653.81,E2 29653.81} C_VEL
LIN {X 0,Y 145.1,Z 1176.161,A -85,B 0,C 180,E1 29660.871,E2 29660.871} C_VEL
LIN {X 0,Y 142.951,Z 1175.855,A -85,B 0,C 180,E1 29663.244,E2 29663.244} C_VEL
LIN {X 0,Y 144.178,Z 1170.453,A -85,B 0,C 180,E1 29704.447,E2 29704.447} C_VEL
LIN {X 0,Y 183.456,Z 1162.834,A -85,B 0,C 180,E1 29721.999,E2 29721.999} C_VEL
LIN {X 0,Y 142.673,Z 1184.211,A -85,B 0,C 180,E1 29739.632,E2 29739.632} C_VEL
LIN {X 0,Y 116.646,Z 1197.021,A -85,B 0,C 180,E1 29771.231,E2 29771.231} C_VEL
LIN {X 0,Y 114.922,Z 1198.646,A -85,B 0,C 180,E1 29793.986,E2 29793.986} C_VEL
LIN {X 0,Y 123.998,Z 1193.085,A -85,B 0,C 180,E1 29823.635,E2 29823.635} C_VEL
LIN {X 0,Y 162.572,Z 1174.54,A -85,B 0,C 180,E1 29850.241,E2 29850.241} C_VEL
LIN {X 0,Y 220.273,Z 1140.72,A -85,B 0,C 180,E1 29865.659,E2 29865.659} C_VEL
LIN {X 0,Y 279.888,Z 1093.188,A -85,B 0,C 180,E1 29873.979,E2 29873.979} C_VEL
LIN {X 0,Y 309.543,Z 1062.651,A -85,B 0,C 180,E1 29877.038,E2 29877.038} C_VEL
LIN {X 0,Y 310.877,Z 1059.147,A -85,B 0,C 180,E1 29881.316,E2 29881.316} C_VEL
LIN {X 0,Y 308.577,Z 1061.357,A -85,B 0,C 180,E1 29884.341,E2 29884.341} C_VEL
LIN {X 0,Y 250.917,Z 1113.406,A -85,B 0,C 180,E1 29890.645,E2 29890.645} C_VEL
LIN {X 0,Y 191.572,Z 1152.673,A -85,B 0,C 180,E1 29901.792,E2 29901.792} C_VEL
LIN {X 0,Y 138.278,Z 1179.69,A -85,B 0,C 180,E1 29924.261,E2 29924.261} C_VEL
LIN {X 0,Y 117.437,Z 1189.506,A -85,B 0,C 180,E1 29950.947,E2 29950.947} C_VEL
LIN {X 0,Y 115.224,Z 1191.093,A -85,B 0,C 180,E1 29973.575,E2 29973.575} C_VEL
LIN {X 0,Y 124.933,Z 1185.834,A -85,B 0,C 180,E1 30002.909,E2 30002.909} C_VEL
LIN {X 0,Y 145.048,Z 1175.97,A -85,B 0,C 180,E1 30021.425,E2 30021.425} C_VEL
LIN {X 0,Y 142.951,Z 1175.855,A -85,B 0,C 180,E1 30023.244,E2 30023.244} C_VEL
LIN {X 0,Y 126.185,Z 1176.909,A -85,B 0,C 180,E1 30036.573,E2 30036.573} C_VEL
LIN {X 0,Y 151.772,Z 1170.506,A -85,B 0,C 180,E1 30074.646,E2 30074.646} C_VEL
LIN {X 0,Y 172.073,Z 1167.257,A -85,B 0,C 180,E1 30082.55,E2 30082.55} C_VEL
LIN {X 0,Y 123.172,Z 1190.142,A -85,B 0,C 180,E1 30107.603,E2 30107.603} C_VEL
LIN {X 0,Y 107.248,Z 1197.842,A -85,B 0,C 180,E1 30137.968,E2 30137.968} C_VEL
LIN {X 0,Y 106.907,Z 1198.381,A -85,B 0,C 180,E1 30154.286,E2 30154.286} C_VEL
LIN {X 0,Y 117.179,Z 1192.794,A -85,B 0,C 180,E1 30185.883,E2 30185.883} C_VEL
LIN {X 0,Y 158.28,Z 1174.294,A -85,B 0,C 180,E1 30212.784,E2 30212.784} C_VEL
LIN {X 0,Y 217.677,Z 1140.654,A -85,B 0,C 180,E1 30227.695,E2 30227.695} C_VEL
LIN {X 0,Y 277.028,Z 1094.436,A -85,B 0,C 180,E1 30235.496,E2 30235.496} C_VEL
LIN {X 0,Y 304.306,Z 1067.46,A -85,B 0,C 180,E1 30238.131,E2 30238.131} C_VEL
LIN {X 0,Y 304.737,Z 1065.351,A -85,B 0,C 180,E1 30242.922,E2 30242.922} C_VEL
LIN {X 0,Y 246.68,Z 1115.958,A -85,B 0,C 180,E1 30249.149,E2 30249.149} C_VEL
LIN {X 0,Y 186.185,Z 1154.353,A -85,B 0,C 180,E1 30260.055,E2 30260.055} C_VEL
LIN {X 0,Y 132.632,Z 1180,A -85,B 0,C 180,E1 30281.699,E2 30281.699} C_VEL
LIN {X 0,Y 109.782,Z 1189.776,A -85,B 0,C 180,E1 30309.561,E2 30309.561} C_VEL
LIN {X 0,Y 107.215,Z 1191.358,A -85,B 0,C 180,E1 30333.842,E2 30333.842} C_VEL
LIN {X 0,Y 121.155,Z 1184.759,A -85,B 0,C 180,E1 30368.526,E2 30368.526} C_VEL
LIN {X 0,Y 134.711,Z 1179.028,A -85,B 0,C 180,E1 30379.683,E2 30379.683} C_VEL
LIN {X 0,Y 135.582,Z 1177.968,A -85,B 0,C 180,E1 30382.251,E2 30382.251} C_VEL
LIN {X 0,Y 126.185,Z 1176.909,A -85,B 0,C 180,E1 30396.573,E2 30396.573} C_VEL
LIN {X 0,Y 119.475,Z 1177.483,A -85,B 0,C 180,E1 30412.854,E2 30412.854} C_VEL
LIN {X 0,Y 160.889,Z 1170.727,A -85,B 0,C 180,E1 30442.13,E2 30442.13} C_VEL
LIN {X 0,Y 115.115,Z 1190.712,A -85,B 0,C 180,E1 30466.784,E2 30466.784} C_VEL
LIN {X 0,Y 99.344,Z 1197.571,A -85,B 0,C 180,E1 30496.994,E2 30496.994} C_VEL
LIN {X 0,Y 98.906,Z 1198.117,A -85,B 0,C 180,E1 30514.633,E2 30514.633} C_VEL
LIN {X 0,Y 110.558,Z 1192.488,A -85,B 0,C 180,E1 30548.407,E2 30548.407} C_VEL
LIN {X 0,Y 154.615,Z 1173.91,A -85,B 0,C 180,E1 30575.556,E2 30575.556} C_VEL
LIN {X 0,Y 216.087,Z 1140.118,A -85,B 0,C 180,E1 30589.907,E2 30589.907} C_VEL
LIN {X 0,Y 277.042,Z 1093.388,A -85,B 0,C 180,E1 30597.287,E2 30597.287} C_VEL
LIN {X 0,Y 299.069,Z 1072.036,A -85,B 0,C 180,E1 30599.561,E2 30599.561} C_VEL
LIN {X 0,Y 298.766,Z 1071.583,A -85,B 0,C 180,E1 30602.018,E2 30602.018} C_VEL
LIN {X 0,Y 238.013,Z 1121.863,A -85,B 0,C 180,E1 30608.184,E2 30608.184} C_VEL
LIN {X 0,Y 173.504,Z 1159.897,A -85,B 0,C 180,E1 30620.068,E2 30620.068} C_VEL
LIN {X 0,Y 118.81,Z 1183.63,A -85,B 0,C 180,E1 30645.106,E2 30645.106} C_VEL
LIN {X 0,Y 99.885,Z 1191.1,A -85,B 0,C 180,E1 30676.591,E2 30676.591} C_VEL
LIN {X 0,Y 99.864,Z 1191.125,A -85,B 0,C 180,E1 30702.937,E2 30702.937} C_VEL
LIN {X 0,Y 123.868,Z 1181.569,A -85,B 0,C 180,E1 30738.651,E2 30738.651} C_VEL
LIN {X 0,Y 126.84,Z 1180.42,A -85,B 0,C 180,E1 30740.75,E2 30740.75} C_VEL
LIN {X 0,Y 119.475,Z 1177.483,A -85,B 0,C 180,E1 30772.854,E2 30772.854} C_VEL
LIN {X 0,Y 124.623,Z 1177.629,A -85,B 0,C 180,E1 30789.371,E2 30789.371} C_VEL
LIN {X 0,Y 149.235,Z 1174.268,A -85,B 0,C 180,E1 30802.025,E2 30802.025} C_VEL
LIN {X 0,Y 103.894,Z 1192.318,A -85,B 0,C 180,E1 30829.206,E2 30829.206} C_VEL
LIN {X 0,Y 90.954,Z 1197.868,A -85,B 0,C 180,E1 30865.47,E2 30865.47} C_VEL
LIN {X 0,Y 96.068,Z 1195.304,A -85,B 0,C 180,E1 30899.159,E2 30899.159} C_VEL
LIN {X 0,Y 135.407,Z 1180.24,A -85,B 0,C 180,E1 30932.462,E2 30932.462} C_VEL
LIN {X 0,Y 195.543,Z 1151.147,A -85,B 0,C 180,E1 30949.024,E2 30949.024} C_VEL
LIN {X 0,Y 258.625,Z 1108.343,A -85,B 0,C 180,E1 30957.354,E2 30957.354} C_VEL
LIN {X 0,Y 293.762,Z 1076.826,A -85,B 0,C 180,E1 30960.806,E2 30960.806} C_VEL
LIN {X 0,Y 232.141,Z 1125.504,A -85,B 0,C 180,E1 30966.784,E2 30966.784} C_VEL
LIN {X 0,Y 167.071,Z 1161.974,A -85,B 0,C 180,E1 30978.372,E2 30978.372} C_VEL
LIN {X 0,Y 113.115,Z 1183.93,A -85,B 0,C 180,E1 31002.155,E2 31002.155} C_VEL
LIN {X 0,Y 92.035,Z 1191.367,A -85,B 0,C 180,E1 31035.423,E2 31035.423} C_VEL
LIN {X 0,Y 91.997,Z 1191.395,A -85,B 0,C 180,E1 31064.065,E2 31064.065} C_VEL
LIN {X 0,Y 117.438,Z 1182.297,A -85,B 0,C 180,E1 31100.889,E2 31100.889} C_VEL
LIN {X 0,Y 124.623,Z 1177.629,A -85,B 0,C 180,E1 31149.371,E2 31149.371} C_VEL
LIN {X 0,Y 132.211,Z 1178.145,A -85,B 0,C 180,E1 31159.526,E2 31159.526} C_VEL
LIN {X 0,Y 137.655,Z 1177.501,A -85,B 0,C 180,E1 31161.835,E2 31161.835} C_VEL
LIN {X 0,Y 91.168,Z 1194.254,A -85,B 0,C 180,E1 31194.683,E2 31194.683} C_VEL
LIN {X 0,Y 82.938,Z 1197.604,A -85,B 0,C 180,E1 31225.031,E2 31225.031} C_VEL
LIN {X 0,Y 86.503,Z 1195.838,A -85,B 0,C 180,E1 31256.307,E2 31256.307} C_VEL
LIN {X 0,Y 127.263,Z 1181.666,A -85,B 0,C 180,E1 31293.815,E2 31293.815} C_VEL
LIN {X 0,Y 190.478,Z 1152.807,A -85,B 0,C 180,E1 31310.869,E2 31310.869} C_VEL
LIN {X 0,Y 256.488,Z 1109.225,A -85,B 0,C 180,E1 31319.057,E2 31319.057} C_VEL
LIN {X 0,Y 273.464,Z 1095.149,A -85,B 0,C 180,E1 31320.761,E2 31320.761} C_VEL
LIN {X 0,Y 207.149,Z 1140.789,A -85,B 0,C 180,E1 31327.778,E2 31327.778} C_VEL
LIN {X 0,Y 140.067,Z 1172.66,A -85,B 0,C 180,E1 31342.53,E2 31342.53} C_VEL
LIN {X 0,Y 92.437,Z 1189.015,A -85,B 0,C 180,E1 31374.629,E2 31374.629} C_VEL
LIN {X 0,Y 83.098,Z 1192.145,A -85,B 0,C 180,E1 31404.483,E2 31404.483} C_VEL
LIN {X 0,Y 87.14,Z 1190.648,A -85,B 0,C 180,E1 31435.512,E2 31435.512} C_VEL
LIN {X 0,Y 109.208,Z 1183.502,A -85,B 0,C 180,E1 31462.861,E2 31462.861} C_VEL
LIN {X 0,Y 127.941,Z 1178.647,A -85,B 0,C 180,E1 31517.455,E2 31517.455} C_VEL
LIN {X 0,Y 132.211,Z 1178.145,A -85,B 0,C 180,E1 31519.526,E2 31519.526} C_VEL
LIN {X 0,Y 127.679,Z 1180.386,A -85,B 0,C 180,E1 31522.921,E2 31522.921} C_VEL
LIN {X 0,Y 114.796,Z 1184.385,A -85,B 0,C 180,E1 31526.642,E2 31526.642} C_VEL
LIN {X 0,Y 79.064,Z 1195.645,A -85,B 0,C 180,E1 31561.661,E2 31561.661} C_VEL
LIN {X 0,Y 74.81,Z 1197.318,A -85,B 0,C 180,E1 31596.131,E2 31596.131} C_VEL
LIN {X 0,Y 95.038,Z 1190.76,A -85,B 0,C 180,E1 31640.55,E2 31640.55} C_VEL
LIN {X 0,Y 152.679,Z 1169.901,A -85,B 0,C 180,E1 31666.313,E2 31666.313} C_VEL
LIN {X 0,Y 220.624,Z 1134.002,A -85,B 0,C 180,E1 31677.515,E2 31677.515} C_VEL
LIN {X 0,Y 250.791,Z 1112.942,A -85,B 0,C 180,E1 31680.852,E2 31680.852} C_VEL
LIN {X 0,Y 184.578,Z 1152.475,A -85,B 0,C 180,E1 31688.642,E2 31688.642} C_VEL
LIN {X 0,Y 119.016,Z 1179.323,A -85,B 0,C 180,E1 31706.26,E2 31706.26} C_VEL
LIN {X 0,Y 80.089,Z 1190.863,A -85,B 0,C 180,E1 31741.402,E2 31741.402} C_VEL
LIN {X 0,Y 75.204,Z 1192.417,A -85,B 0,C 180,E1 31775.482,E2 31775.482} C_VEL
LIN {X 0,Y 97.541,Z 1185.969,A -85,B 0,C 180,E1 31820.612,E2 31820.612} C_VEL
LIN {X 0,Y 98.204,Z 1184.908,A -85,B 0,C 180,E1 31827.573,E2 31827.573} C_VEL
LIN {X 0,Y 125.446,Z 1180.431,A -85,B 0,C 180,E1 31881.35,E2 31881.35} C_VEL
LIN {X 0,Y 114.796,Z 1184.385,A -85,B 0,C 180,E1 31886.642,E2 31886.642} C_VEL
LIN {X 0,Y 86.567,Z 1191.433,A -85,B 0,C 180,E1 31898.37,E2 31898.37} C_VEL
LIN {X 0,Y 66.883,Z 1197.074,A -85,B 0,C 180,E1 31943.834,E2 31943.834} C_VEL
LIN {X 0,Y 72.175,Z 1195.289,A -85,B 0,C 180,E1 31982.083,E2 31982.083} C_VEL
LIN {X 0,Y 120.774,Z 1180.984,A -85,B 0,C 180,E1 32021.013,E2 32021.013} C_VEL
LIN {X 0,Y 187.6,Z 1152.372,A -85,B 0,C 180,E1 32035.852,E2 32035.852} C_VEL
LIN {X 0,Y 228.581,Z 1128.267,A -85,B 0,C 180,E1 32040.466,E2 32040.466} C_VEL
LIN {X 0,Y 159.455,Z 1163.701,A -85,B 0,C 180,E1 32050.243,E2 32050.243} C_VEL
LIN {X 0,Y 94.403,Z 1185.8,A -85,B 0,C 180,E1 32073.904,E2 32073.904} C_VEL
LIN {X 0,Y 68.809,Z 1192.165,A -85,B 0,C 180,E1 32110.329,E2 32110.329} C_VEL
LIN {X 0,Y 67.217,Z 1192.681,A -85,B 0,C 180,E1 32136.135,E2 32136.135} C_VEL
LIN {X 0,Y 87.725,Z 1187.556,A -85,B 0,C 180,E1 32180.692,E2 32180.692} C_VEL
LIN {X 0,Y 91.402,Z 1186.414,A -85,B 0,C 180,E1 32184.822,E2 32184.822} C_VEL
LIN {X 0,Y 113.991,Z 1183.031,A -85,B 0,C 180,E1 32241.017,E2 32241.017} C_VEL
LIN {X 0,Y 86.567,Z 1191.433,A -85,B 0,C 180,E1 32258.37,E2 32258.37} C_VEL
LIN {X 0,Y 63.274,Z 1195.481,A -85,B 0,C 180,E1 32278.94,E2 32278.94} C_VEL
LIN {X 0,Y 58.787,Z 1196.787,A -85,B 0,C 180,E1 32317.811,E2 32317.811} C_VEL
LIN {X 0,Y 82.176,Z 1191.015,A -85,B 0,C 180,E1 32366.699,E2 32366.699} C_VEL
LIN {X 0,Y 146.01,Z 1170.665,A -85,B 0,C 180,E1 32391.891,E2 32391.891} C_VEL
LIN {X 0,Y 205.267,Z 1142.116,A -85,B 0,C 180,E1 32400.884,E2 32400.884} C_VEL
LIN {X 0,Y 132.536,Z 1173.704,A -85,B 0,C 180,E1 32412.537,E2 32412.537} C_VEL
LIN {X 0,Y 73.775,Z 1189.856,A -85,B 0,C 180,E1 32443.506,E2 32443.506} C_VEL
LIN {X 0,Y 59.117,Z 1192.94,A -85,B 0,C 180,E1 32482.233,E2 32482.233} C_VEL
LIN {X 0,Y 69.401,Z 1190.743,A -85,B 0,C 180,E1 32530.645,E2 32530.645} C_VEL
LIN {X 0,Y 82.519,Z 1187.861,A -85,B 0,C 180,E1 32545.343,E2 32545.343} C_VEL
LIN {X 0,Y 102.594,Z 1185.381,A -85,B 0,C 180,E1 32600.528,E2 32600.528} C_VEL
LIN {X 0,Y 63.274,Z 1195.481,A -85,B 0,C 180,E1 32638.94,E2 32638.94} C_VEL
LIN {X 0,Y 50.312,Z 1196.528,A -85,B 0,C 180,E1 32673.234,E2 32673.234} C_VEL
LIN {X 0,Y 73.899,Z 1191.656,A -85,B 0,C 180,E1 32728.714,E2 32728.714} C_VEL
LIN {X 0,Y 141.31,Z 1171.658,A -85,B 0,C 180,E1 32754.525,E2 32754.525} C_VEL
LIN {X 0,Y 182.778,Z 1153.655,A -85,B 0,C 180,E1 32760.55,E2 32760.55} C_VEL
LIN {X 0,Y 116.966,Z 1178.44,A -85,B 0,C 180,E1 32772.478,E2 32772.478} C_VEL
LIN {X 0,Y 59.791,Z 1191.689,A -85,B 0,C 180,E1 32810.121,E2 32810.121} C_VEL
LIN {X 0,Y 51.237,Z 1193.21,A -85,B 0,C 180,E1 32858.06,E2 32858.06} C_VEL
LIN {X 0,Y 72.769,Z 1189.227,A -85,B 0,C 180,E1 32905.753,E2 32905.753} C_VEL
LIN {X 0,Y 90.651,Z 1187.415,A -85,B 0,C 180,E1 32959.572,E2 32959.572} C_VEL
LIN {X 0,Y 55.728,Z 1195.295,A -85,B 0,C 180,E1 32996.164,E2 32996.164} C_VEL
LIN {X 0,Y 50.312,Z 1196.528,A -85,B 0,C 180,E1 33033.234,E2 33033.234} C_VEL
LIN {X 0,Y 51.592,Z 1194.667,A -85,B 0,C 180,E1 33074.181,E2 33074.181} C_VEL
LIN {X 0,Y 112.088,Z 1180.867,A -85,B 0,C 180,E1 33112.284,E2 33112.284} C_VEL
LIN {X 0,Y 159.741,Z 1163.845,A -85,B 0,C 180,E1 33120.873,E2 33120.873} C_VEL
LIN {X 0,Y 87.897,Z 1185.713,A -85,B 0,C 180,E1 33137.442,E2 33137.442} C_VEL
LIN {X 0,Y 46.62,Z 1192.977,A -85,B 0,C 180,E1 33180.209,E2 33180.209} C_VEL
LIN {X 0,Y 43.269,Z 1193.476,A -85,B 0,C 180,E1 33219.557,E2 33219.557} C_VEL
LIN {X 0,Y 64.308,Z 1190.272,A -85,B 0,C 180,E1 33267.829,E2 33267.829} C_VEL
LIN {X 0,Y 79.365,Z 1189.185,A -85,B 0,C 180,E1 33318.734,E2 33318.734} C_VEL
LIN {X 0,Y 45.723,Z 1195.679,A -85,B 0,C 180,E1 33360.727,E2 33360.727} C_VEL
LIN {X 0,Y 42.828,Z 1196.255,A -85,B 0,C 180,E1 33400.751,E2 33400.751} C_VEL
LIN {X 0,Y 51.592,Z 1194.667,A -85,B 0,C 180,E1 33434.181,E2 33434.181} C_VEL
LIN {X 0,Y 70.309,Z 1190.345,A -85,B 0,C 180,E1 33463.012,E2 33463.012} C_VEL
LIN {X 0,Y 135.982,Z 1172.608,A -85,B 0,C 180,E1 33480.745,E2 33480.745} C_VEL
LIN {X 0,Y 65.628,Z 1189.723,A -85,B 0,C 180,E1 33501.701,E2 33501.701} C_VEL
LIN {X 0,Y 35.324,Z 1193.735,A -85,B 0,C 180,E1 33556.928,E2 33556.928} C_VEL
LIN {X 0,Y 47.901,Z 1192.292,A -85,B 0,C 180,E1 33621.583,E2 33621.583} C_VEL
LIN {X 0,Y 54.895,Z 1191.379,A -85,B 0,C 180,E1 33629.764,E2 33629.764} C_VEL
LIN {X 0,Y 67.463,Z 1190.752,A -85,B 0,C 180,E1 33676.722,E2 33676.722} C_VEL
LIN {X 0,Y 38.83,Z 1195.411,A -85,B 0,C 180,E1 33714.846,E2 33714.846} C_VEL
LIN {X 0,Y 34.906,Z 1195.988,A -85,B 0,C 180,E1 33763.231,E2 33763.231} C_VEL
LIN {X 0,Y 70.309,Z 1190.345,A -85,B 0,C 180,E1 33823.012,E2 33823.012} C_VEL
LIN {X 0,Y 97.432,Z 1183.822,A -85,B 0,C 180,E1 33838.32,E2 33838.32} C_VEL
LIN {X 0,Y 108.574,Z 1180.874,A -85,B 0,C 180,E1 33840.48,E2 33840.48} C_VEL
LIN {X 0,Y 56.427,Z 1190.975,A -85,B 0,C 180,E1 33858.507,E2 33858.507} C_VEL
LIN {X 0,Y 27.526,Z 1194,A -85,B 0,C 180,E1 33913.127,E2 33913.127} C_VEL
LIN {X 0,Y 45.973,Z 1192.257,A -85,B 0,C 180,E1 33993.022,E2 33993.022} C_VEL
LIN {X 0,Y 56.501,Z 1191.951,A -85,B 0,C 180,E1 34035.096,E2 34035.096} C_VEL
LIN {X 0,Y 27.046,Z 1195.742,A -85,B 0,C 180,E1 34094.596,E2 34094.596} C_VEL
LIN {X 0,Y 43.25,Z 1193.9,A -85,B 0,C 180,E1 34172.421,E2 34172.421} C_VEL
LIN {X 0,Y 97.432,Z 1183.822,A -85,B 0,C 180,E1 34198.32,E2 34198.32} C_VEL
LIN {X 0,Y 74.933,Z 1188.193,A -85,B 0,C 180,E1 34203.094,E2 34203.094} C_VEL
LIN {X 0,Y 19.94,Z 1194.266,A -85,B 0,C 180,E1 34266.38,E2 34266.38} C_VEL
LIN {X 0,Y 38.327,Z 1192.996,A -85,B 0,C 180,E1 34358.84,E2 34358.84} C_VEL
LIN {X 0,Y 45.345,Z 1192.953,A -85,B 0,C 180,E1 34392.015,E2 34392.015} C_VEL
LIN {X 0,Y 19.366,Z 1195.476,A -85,B 0,C 180,E1 34448.225,E2 34448.225} C_VEL
LIN {X 0,Y 40.102,Z 1193.625,A -85,B 0,C 180,E1 34542.933,E2 34542.933} C_VEL
LIN {X 0,Y 83.869,Z 1186.619,A -85,B 0,C 180,E1 34560.993,E2 34560.993} C_VEL
LIN {X 0,Y 74.933,Z 1188.193,A -85,B 0,C 180,E1 34563.094,E2 34563.094} C_VEL
LIN {X 0,Y 39.885,Z 1192.934,A -85,B 0,C 180,E1 34566.822,E2 34566.822} C_VEL
LIN {X 0,Y 12.629,Z 1194.539,A -85,B 0,C 180,E1 34684.67,E2 34684.67} C_VEL
LIN {X 0,Y 31.563,Z 1193.671,A -85,B 0,C 180,E1 34730.435,E2 34730.435} C_VEL
LIN {X 0,Y 33.982,Z 1193.743,A -85,B 0,C 180,E1 34745.047,E2 34745.047} C_VEL
LIN {X 0,Y 12.211,Z 1195.207,A -85,B 0,C 180,E1 34793.961,E2 34793.961} C_VEL
LIN {X 0,Y 38.497,Z 1193.35,A -85,B 0,C 180,E1 34914.758,E2 34914.758} C_VEL
LIN {X 0,Y 53.529,Z 1191.55,A -85,B 0,C 180,E1 34921.564,E2 34921.564} C_VEL
LIN {X 0,Y 39.885,Z 1192.934,A -85,B 0,C 180,E1 34926.822,E2 34926.822} C_VEL
LIN {X 0,Y 16.178,Z 1194.661,A -85,B 0,C 180,E1 34919.344,E2 34919.344} C_VEL
LIN {X 0,Y 18.083,Z 1194.598,A -85,B 0,C 180,E1 34739.712,E2 34739.712} C_VEL
LIN {X 0,Y 8.265,Z 1194.8,A -85,B 0,C 180,E1 34574.837,E2 34574.837} C_VEL
LIN {X 0,Y 18.422,Z 1194.59,A -85,B 0,C 180,E1 34560.618,E2 34560.618} C_VEL
LIN {X 0,Y 16.178,Z 1194.661,A -85,B 0,C 180,E1 34559.344,E2 34559.344} C_VEL
LIN {X 0,Y 14.277,Z 1196.66,A -85,B 0,C 180,E1 34557.945,E2 34557.945} C_VEL
LIN {X 0,Y 14.277,Z 1215,A -85,B 0,C 180,E1 34557.945,E2 34557.945} C_VEL
LIN {X 0,Y 14.277,Z 1215,A -85,B 0,C 180,E1 34557.945,E2 34557.945}

